// TIA Portal V17 export
// export: Created 2025-04-09T08:03:29.2675501Z, ExportSetting WithDefaults, DisplayName Totally Integrated Automation Portal, DisplayVersion V17 Update 8, DisplayName TIA Portal Openness, DisplayVersion V17 Update 8, DisplayName TIA Portal Version Control Interface, DisplayVersion V17, DisplayName SINAMICS Startdrive Advanced, DisplayVersion V17 SP2, DisplayName SINAMICS Startdrive G110M, G120, G120C, G120D, G120P, G115D, DisplayVersion V17 SP2, DisplayName SINAMICS Startdrive G130, G150, S120, S150, SINAMICS MV, S210, DisplayVersion V17 SP2, DisplayName STEP 7 Professional, DisplayVersion V17 Update 8, DisplayName SINUMERIK ONE STEP 7 Toolbox, DisplayVersion V17 Update 12, DisplayName SINUMERIK ONE PLC Basic Program Plus, DisplayVersion V17 Update 12, DisplayName SINUMERIK 840D sl STEP 7 Toolbox, DisplayVersion V17 Update 12, DisplayName STEP 7 Safety, DisplayVersion V17 Update 6, DisplayName WinCC Advanced, DisplayVersion V17 Update 8
FUNCTION "FC16012_METHOD_CALLS_U01_STA3_COAXIAL" : Void   // FC16012, LAD
{ S7_Optimized_Access := 'TRUE' }
VERSION : 0.1
// PC status values:
// 0-> Idle
// 1-> LaserCalibrating
// 2-> NozzleCalibrating
// 3-> JetCalibrating
// 4-> CladdingCalibrating
// 5-> NozzleAnalysis
// 6-> JetAnalysis
// 7-> CladdingAnalysis
// -1-> Error
// stored: AutoNumber false, IsIECCheckEnabled false, SetENOAutomatically false, UDAEnableTagReadback false
   VAR_TEMP
      AUX_WSTRING_PART_ID_STA3 : WString;
      AUX_WCHARS : Array[0..63] of WChar;
      index : Int;
      ALARM_AUX : Bool;
   END_VAR
   VAR CONSTANT
      VERSIONS_MAJOR : UInt;
      VERSIONS_MINOR : UInt;
      FC_NUMBER : DInt := 16012;
   END_VAR
   VAR_TEMP   // added for the SCL form of the ladder/FBD networks
      _w1 : Bool;
      _w2 : Bool;
   END_VAR
BEGIN

REGION Network 1 (SCL): TRANSFORM TO WCHARS
   FOR #index := 0 TO 63 DO
       #AUX_WCHARS[#index] := CHAR_TO_WCHAR("DB8000_PART_STATUS".UNIT_01.STATION_3.PART_A.PART_ID[#index]);
   END_FOR;
END_REGION

REGION Network 2: TRANSFORM TO WSTRING
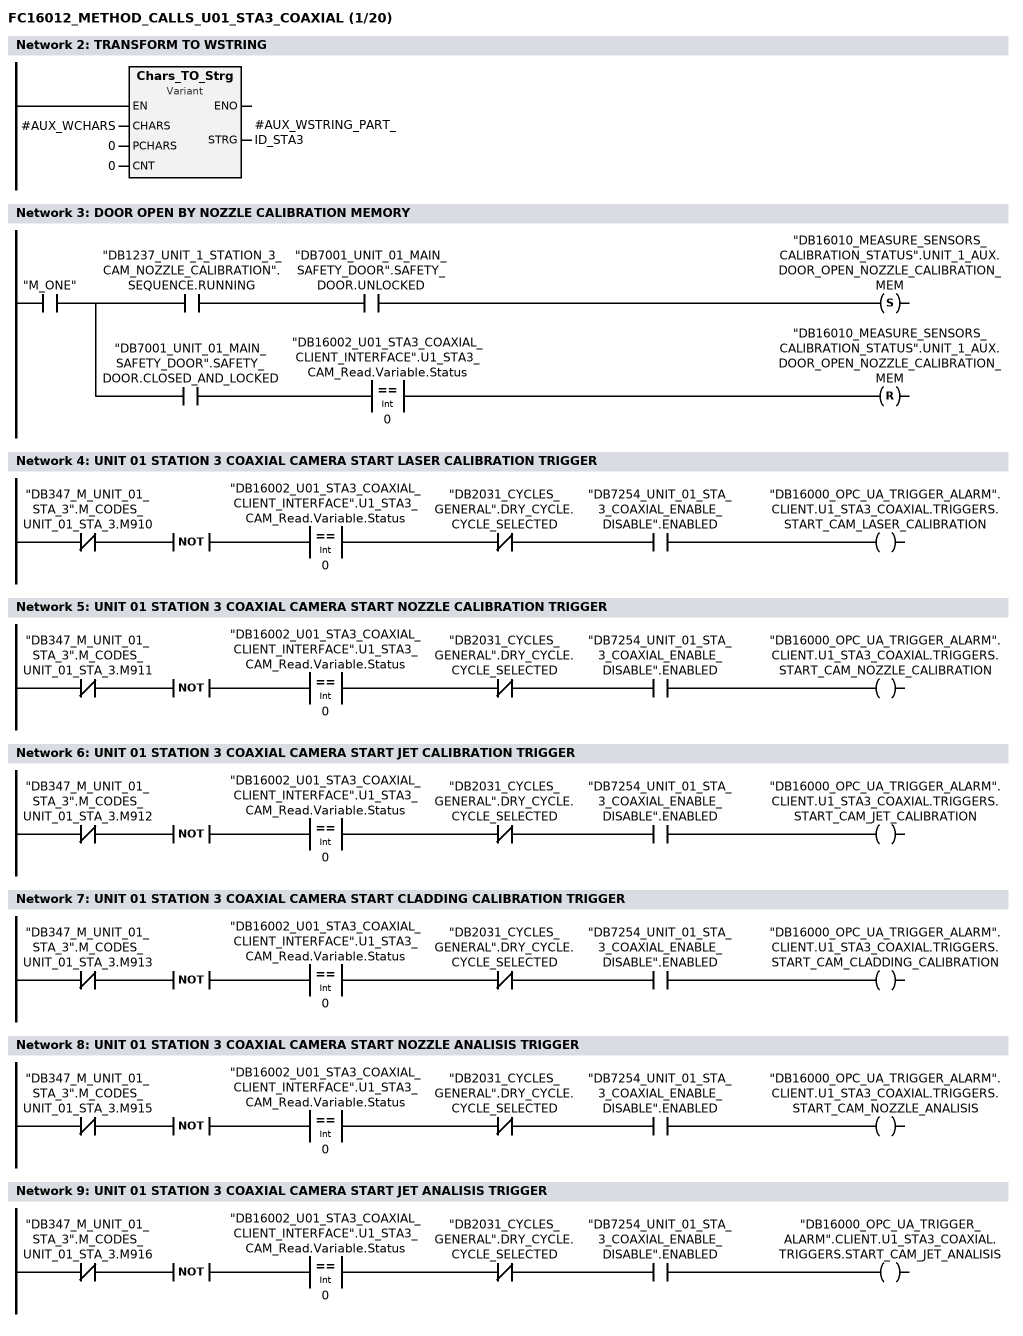
   RUNG wire#powerrail
      { S7_Templates := "[ptr_type := Variant, str_type := WString]" } Chars_TO_Strg(Chars := #AUX_WCHARS, pChars := 0, Cnt := 0, Strg => #AUX_WSTRING_PART_ID_STA3)
   END_RUNG
   // the same network as SCL:
   Chars_TO_Strg(Chars := #AUX_WCHARS, pChars := 0, Cnt := 0, Strg => #AUX_WSTRING_PART_ID_STA3);
END_REGION

REGION Network 3: DOOR OPEN BY NOZZLE CALIBRATION MEMORY
   RUNG wire#powerrail
      Contact( "M_ONE" )
      wire#w1
      Contact( "DB1237_UNIT_1_STATION_3_CAM_NOZZLE_CALIBRATION".SEQUENCE.RUNNING )
      Contact( "DB7001_UNIT_01_MAIN_SAFETY_DOOR".SAFETY_DOOR.UNLOCKED )
      S_Coil( "DB16010_MEASURE_SENSORS_CALIBRATION_STATUS".UNIT_1_AUX.DOOR_OPEN_NOZZLE_CALIBRATION_MEM )
   END_RUNG
   RUNG wire#w1
      Contact( "DB7001_UNIT_01_MAIN_SAFETY_DOOR".SAFETY_DOOR.CLOSED_AND_LOCKED )
      { S7_Templates := "SrcType := Int" } EQ_Contact(in1 := "DB16002_U01_STA3_COAXIAL_CLIENT_INTERFACE".U1_STA3_CAM_Read.Variable.Status, in2 := 0)
      R_Coil( "DB16010_MEASURE_SENSORS_CALIBRATION_STATUS".UNIT_1_AUX.DOOR_OPEN_NOZZLE_CALIBRATION_MEM )
   END_RUNG
   // the same network as SCL:
   IF "M_ONE" AND "DB1237_UNIT_1_STATION_3_CAM_NOZZLE_CALIBRATION".SEQUENCE.RUNNING AND "DB7001_UNIT_01_MAIN_SAFETY_DOOR".SAFETY_DOOR.UNLOCKED THEN
       "DB16010_MEASURE_SENSORS_CALIBRATION_STATUS".UNIT_1_AUX.DOOR_OPEN_NOZZLE_CALIBRATION_MEM := TRUE;
   END_IF;
   IF "M_ONE" AND "DB7001_UNIT_01_MAIN_SAFETY_DOOR".SAFETY_DOOR.CLOSED_AND_LOCKED AND ("DB16002_U01_STA3_COAXIAL_CLIENT_INTERFACE".U1_STA3_CAM_Read.Variable.Status = 0) THEN
       "DB16010_MEASURE_SENSORS_CALIBRATION_STATUS".UNIT_1_AUX.DOOR_OPEN_NOZZLE_CALIBRATION_MEM := FALSE;
   END_IF;
END_REGION

REGION Network 4: UNIT 01 STATION 3 COAXIAL CAMERA START LASER CALIBRATION TRIGGER
   RUNG wire#powerrail
      I_Contact( "DB347_M_UNIT_01_STA_3".M_CODES_UNIT_01_STA_3.M910 )
      Not()
      { S7_Templates := "SrcType := Int" } EQ_Contact(in1 := "DB16002_U01_STA3_COAXIAL_CLIENT_INTERFACE".U1_STA3_CAM_Read.Variable.Status, in2 := 0)
      I_Contact( "DB2031_CYCLES_GENERAL".DRY_CYCLE.CYCLE_SELECTED )
      Contact( "DB7254_UNIT_01_STA_3_COAXIAL_ENABLE_DISABLE".ENABLED )
      Coil( "DB16000_OPC_UA_TRIGGER_ALARM".CLIENT.U1_STA3_COAXIAL.TRIGGERS.START_CAM_LASER_CALIBRATION )
   END_RUNG
   // the same network as SCL:
   "DB16000_OPC_UA_TRIGGER_ALARM".CLIENT.U1_STA3_COAXIAL.TRIGGERS.START_CAM_LASER_CALIBRATION := NOT (NOT "DB347_M_UNIT_01_STA_3".M_CODES_UNIT_01_STA_3.M910) AND ("DB16002_U01_STA3_COAXIAL_CLIENT_INTERFACE".U1_STA3_CAM_Read.Variable.Status = 0) AND NOT "DB2031_CYCLES_GENERAL".DRY_CYCLE.CYCLE_SELECTED AND "DB7254_UNIT_01_STA_3_COAXIAL_ENABLE_DISABLE".ENABLED;
END_REGION

REGION Network 5: UNIT 01 STATION 3 COAXIAL CAMERA START NOZZLE CALIBRATION TRIGGER
   RUNG wire#powerrail
      I_Contact( "DB347_M_UNIT_01_STA_3".M_CODES_UNIT_01_STA_3.M911 )
      Not()
      { S7_Templates := "SrcType := Int" } EQ_Contact(in1 := "DB16002_U01_STA3_COAXIAL_CLIENT_INTERFACE".U1_STA3_CAM_Read.Variable.Status, in2 := 0)
      I_Contact( "DB2031_CYCLES_GENERAL".DRY_CYCLE.CYCLE_SELECTED )
      Contact( "DB7254_UNIT_01_STA_3_COAXIAL_ENABLE_DISABLE".ENABLED )
      Coil( "DB16000_OPC_UA_TRIGGER_ALARM".CLIENT.U1_STA3_COAXIAL.TRIGGERS.START_CAM_NOZZLE_CALIBRATION )
   END_RUNG
   // the same network as SCL:
   "DB16000_OPC_UA_TRIGGER_ALARM".CLIENT.U1_STA3_COAXIAL.TRIGGERS.START_CAM_NOZZLE_CALIBRATION := NOT (NOT "DB347_M_UNIT_01_STA_3".M_CODES_UNIT_01_STA_3.M911) AND ("DB16002_U01_STA3_COAXIAL_CLIENT_INTERFACE".U1_STA3_CAM_Read.Variable.Status = 0) AND NOT "DB2031_CYCLES_GENERAL".DRY_CYCLE.CYCLE_SELECTED AND "DB7254_UNIT_01_STA_3_COAXIAL_ENABLE_DISABLE".ENABLED;
END_REGION

REGION Network 6: UNIT 01 STATION 3 COAXIAL CAMERA START JET CALIBRATION TRIGGER
   RUNG wire#powerrail
      I_Contact( "DB347_M_UNIT_01_STA_3".M_CODES_UNIT_01_STA_3.M912 )
      Not()
      { S7_Templates := "SrcType := Int" } EQ_Contact(in1 := "DB16002_U01_STA3_COAXIAL_CLIENT_INTERFACE".U1_STA3_CAM_Read.Variable.Status, in2 := 0)
      I_Contact( "DB2031_CYCLES_GENERAL".DRY_CYCLE.CYCLE_SELECTED )
      Contact( "DB7254_UNIT_01_STA_3_COAXIAL_ENABLE_DISABLE".ENABLED )
      Coil( "DB16000_OPC_UA_TRIGGER_ALARM".CLIENT.U1_STA3_COAXIAL.TRIGGERS.START_CAM_JET_CALIBRATION )
   END_RUNG
   // the same network as SCL:
   "DB16000_OPC_UA_TRIGGER_ALARM".CLIENT.U1_STA3_COAXIAL.TRIGGERS.START_CAM_JET_CALIBRATION := NOT (NOT "DB347_M_UNIT_01_STA_3".M_CODES_UNIT_01_STA_3.M912) AND ("DB16002_U01_STA3_COAXIAL_CLIENT_INTERFACE".U1_STA3_CAM_Read.Variable.Status = 0) AND NOT "DB2031_CYCLES_GENERAL".DRY_CYCLE.CYCLE_SELECTED AND "DB7254_UNIT_01_STA_3_COAXIAL_ENABLE_DISABLE".ENABLED;
END_REGION

REGION Network 7: UNIT 01 STATION 3 COAXIAL CAMERA START CLADDING CALIBRATION TRIGGER
   RUNG wire#powerrail
      I_Contact( "DB347_M_UNIT_01_STA_3".M_CODES_UNIT_01_STA_3.M913 )
      Not()
      { S7_Templates := "SrcType := Int" } EQ_Contact(in1 := "DB16002_U01_STA3_COAXIAL_CLIENT_INTERFACE".U1_STA3_CAM_Read.Variable.Status, in2 := 0)
      I_Contact( "DB2031_CYCLES_GENERAL".DRY_CYCLE.CYCLE_SELECTED )
      Contact( "DB7254_UNIT_01_STA_3_COAXIAL_ENABLE_DISABLE".ENABLED )
      Coil( "DB16000_OPC_UA_TRIGGER_ALARM".CLIENT.U1_STA3_COAXIAL.TRIGGERS.START_CAM_CLADDING_CALIBRATION )
   END_RUNG
   // the same network as SCL:
   "DB16000_OPC_UA_TRIGGER_ALARM".CLIENT.U1_STA3_COAXIAL.TRIGGERS.START_CAM_CLADDING_CALIBRATION := NOT (NOT "DB347_M_UNIT_01_STA_3".M_CODES_UNIT_01_STA_3.M913) AND ("DB16002_U01_STA3_COAXIAL_CLIENT_INTERFACE".U1_STA3_CAM_Read.Variable.Status = 0) AND NOT "DB2031_CYCLES_GENERAL".DRY_CYCLE.CYCLE_SELECTED AND "DB7254_UNIT_01_STA_3_COAXIAL_ENABLE_DISABLE".ENABLED;
END_REGION

REGION Network 8: UNIT 01 STATION 3 COAXIAL CAMERA START NOZZLE ANALISIS TRIGGER
   RUNG wire#powerrail
      I_Contact( "DB347_M_UNIT_01_STA_3".M_CODES_UNIT_01_STA_3.M915 )
      Not()
      { S7_Templates := "SrcType := Int" } EQ_Contact(in1 := "DB16002_U01_STA3_COAXIAL_CLIENT_INTERFACE".U1_STA3_CAM_Read.Variable.Status, in2 := 0)
      I_Contact( "DB2031_CYCLES_GENERAL".DRY_CYCLE.CYCLE_SELECTED )
      Contact( "DB7254_UNIT_01_STA_3_COAXIAL_ENABLE_DISABLE".ENABLED )
      Coil( "DB16000_OPC_UA_TRIGGER_ALARM".CLIENT.U1_STA3_COAXIAL.TRIGGERS.START_CAM_NOZZLE_ANALISIS )
   END_RUNG
   // the same network as SCL:
   "DB16000_OPC_UA_TRIGGER_ALARM".CLIENT.U1_STA3_COAXIAL.TRIGGERS.START_CAM_NOZZLE_ANALISIS := NOT (NOT "DB347_M_UNIT_01_STA_3".M_CODES_UNIT_01_STA_3.M915) AND ("DB16002_U01_STA3_COAXIAL_CLIENT_INTERFACE".U1_STA3_CAM_Read.Variable.Status = 0) AND NOT "DB2031_CYCLES_GENERAL".DRY_CYCLE.CYCLE_SELECTED AND "DB7254_UNIT_01_STA_3_COAXIAL_ENABLE_DISABLE".ENABLED;
END_REGION

REGION Network 9: UNIT 01 STATION 3 COAXIAL CAMERA START JET ANALISIS TRIGGER
   RUNG wire#powerrail
      I_Contact( "DB347_M_UNIT_01_STA_3".M_CODES_UNIT_01_STA_3.M916 )
      Not()
      { S7_Templates := "SrcType := Int" } EQ_Contact(in1 := "DB16002_U01_STA3_COAXIAL_CLIENT_INTERFACE".U1_STA3_CAM_Read.Variable.Status, in2 := 0)
      I_Contact( "DB2031_CYCLES_GENERAL".DRY_CYCLE.CYCLE_SELECTED )
      Contact( "DB7254_UNIT_01_STA_3_COAXIAL_ENABLE_DISABLE".ENABLED )
      Coil( "DB16000_OPC_UA_TRIGGER_ALARM".CLIENT.U1_STA3_COAXIAL.TRIGGERS.START_CAM_JET_ANALISIS )
   END_RUNG
   // the same network as SCL:
   "DB16000_OPC_UA_TRIGGER_ALARM".CLIENT.U1_STA3_COAXIAL.TRIGGERS.START_CAM_JET_ANALISIS := NOT (NOT "DB347_M_UNIT_01_STA_3".M_CODES_UNIT_01_STA_3.M916) AND ("DB16002_U01_STA3_COAXIAL_CLIENT_INTERFACE".U1_STA3_CAM_Read.Variable.Status = 0) AND NOT "DB2031_CYCLES_GENERAL".DRY_CYCLE.CYCLE_SELECTED AND "DB7254_UNIT_01_STA_3_COAXIAL_ENABLE_DISABLE".ENABLED;
END_REGION

REGION Network 10: UNIT 01 STATION 3 COAXIAL CAMERA START CLADDING ANALISIS TRIGGER
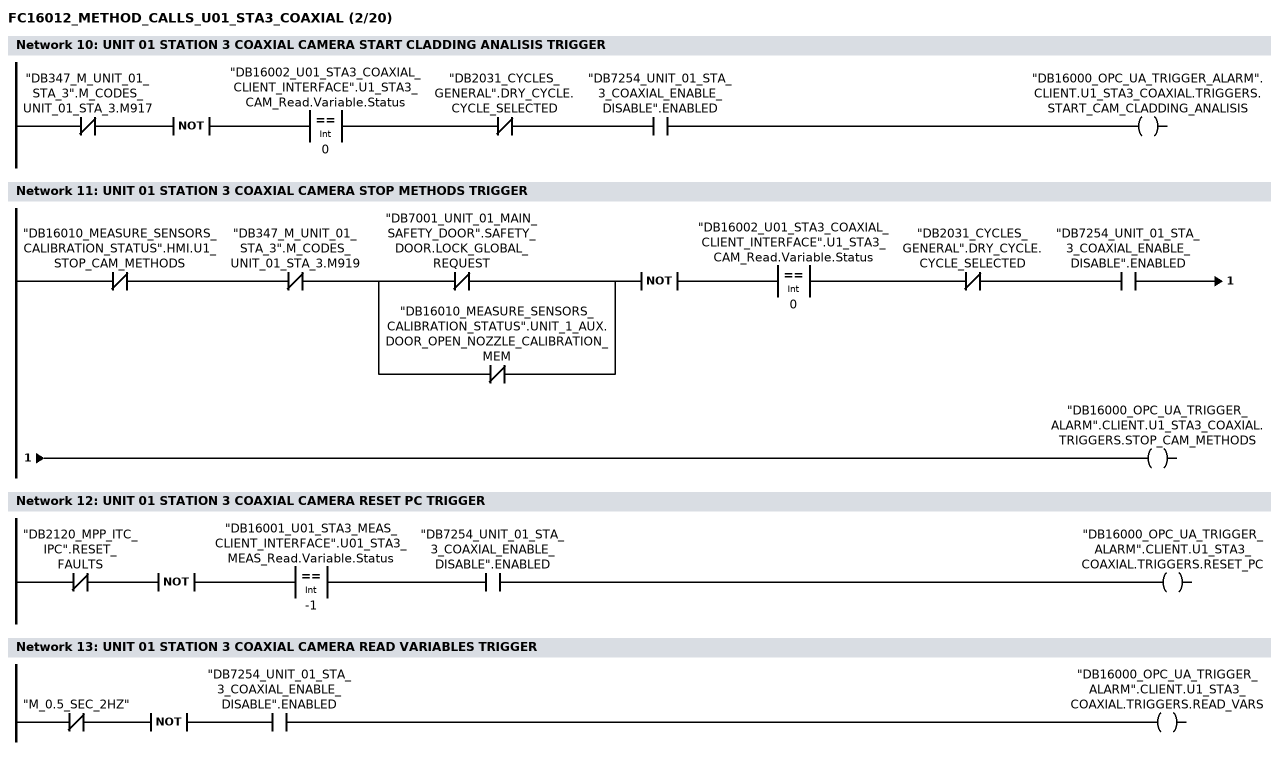
   RUNG wire#powerrail
      I_Contact( "DB347_M_UNIT_01_STA_3".M_CODES_UNIT_01_STA_3.M917 )
      Not()
      { S7_Templates := "SrcType := Int" } EQ_Contact(in1 := "DB16002_U01_STA3_COAXIAL_CLIENT_INTERFACE".U1_STA3_CAM_Read.Variable.Status, in2 := 0)
      I_Contact( "DB2031_CYCLES_GENERAL".DRY_CYCLE.CYCLE_SELECTED )
      Contact( "DB7254_UNIT_01_STA_3_COAXIAL_ENABLE_DISABLE".ENABLED )
      Coil( "DB16000_OPC_UA_TRIGGER_ALARM".CLIENT.U1_STA3_COAXIAL.TRIGGERS.START_CAM_CLADDING_ANALISIS )
   END_RUNG
   // the same network as SCL:
   "DB16000_OPC_UA_TRIGGER_ALARM".CLIENT.U1_STA3_COAXIAL.TRIGGERS.START_CAM_CLADDING_ANALISIS := NOT (NOT "DB347_M_UNIT_01_STA_3".M_CODES_UNIT_01_STA_3.M917) AND ("DB16002_U01_STA3_COAXIAL_CLIENT_INTERFACE".U1_STA3_CAM_Read.Variable.Status = 0) AND NOT "DB2031_CYCLES_GENERAL".DRY_CYCLE.CYCLE_SELECTED AND "DB7254_UNIT_01_STA_3_COAXIAL_ENABLE_DISABLE".ENABLED;
END_REGION

REGION Network 11: UNIT 01 STATION 3 COAXIAL CAMERA STOP METHODS TRIGGER
   RUNG wire#powerrail
      I_Contact( "DB16010_MEASURE_SENSORS_CALIBRATION_STATUS".HMI.U1_STOP_CAM_METHODS )
      I_Contact( "DB347_M_UNIT_01_STA_3".M_CODES_UNIT_01_STA_3.M919 )
      wire#w1
      I_Contact( "DB7001_UNIT_01_MAIN_SAFETY_DOOR".SAFETY_DOOR.LOCK_GLOBAL_REQUEST )
      wire#w2
      Not()
      { S7_Templates := "SrcType := Int" } EQ_Contact(in1 := "DB16002_U01_STA3_COAXIAL_CLIENT_INTERFACE".U1_STA3_CAM_Read.Variable.Status, in2 := 0)
      I_Contact( "DB2031_CYCLES_GENERAL".DRY_CYCLE.CYCLE_SELECTED )
      Contact( "DB7254_UNIT_01_STA_3_COAXIAL_ENABLE_DISABLE".ENABLED )
      Coil( "DB16000_OPC_UA_TRIGGER_ALARM".CLIENT.U1_STA3_COAXIAL.TRIGGERS.STOP_CAM_METHODS )
   END_RUNG
   RUNG wire#w1
      I_Contact( "DB16010_MEASURE_SENSORS_CALIBRATION_STATUS".UNIT_1_AUX.DOOR_OPEN_NOZZLE_CALIBRATION_MEM )
   END_RUNG wire#w2
   // the same network as SCL:
   "DB16000_OPC_UA_TRIGGER_ALARM".CLIENT.U1_STA3_COAXIAL.TRIGGERS.STOP_CAM_METHODS := NOT (NOT "DB16010_MEASURE_SENSORS_CALIBRATION_STATUS".HMI.U1_STOP_CAM_METHODS AND NOT "DB347_M_UNIT_01_STA_3".M_CODES_UNIT_01_STA_3.M919 AND (NOT "DB7001_UNIT_01_MAIN_SAFETY_DOOR".SAFETY_DOOR.LOCK_GLOBAL_REQUEST OR NOT "DB16010_MEASURE_SENSORS_CALIBRATION_STATUS".UNIT_1_AUX.DOOR_OPEN_NOZZLE_CALIBRATION_MEM)) AND ("DB16002_U01_STA3_COAXIAL_CLIENT_INTERFACE".U1_STA3_CAM_Read.Variable.Status = 0) AND NOT "DB2031_CYCLES_GENERAL".DRY_CYCLE.CYCLE_SELECTED AND "DB7254_UNIT_01_STA_3_COAXIAL_ENABLE_DISABLE".ENABLED;
END_REGION

REGION Network 12: UNIT 01 STATION 3 COAXIAL CAMERA RESET PC TRIGGER
   RUNG wire#powerrail
      I_Contact( "DB2120_MPP_ITC_IPC".RESET_FAULTS )
      Not()
      { S7_Templates := "SrcType := Int" } EQ_Contact(in1 := "DB16001_U01_STA3_MEAS_CLIENT_INTERFACE".U01_STA3_MEAS_Read.Variable.Status, in2 := -1)
      Contact( "DB7254_UNIT_01_STA_3_COAXIAL_ENABLE_DISABLE".ENABLED )
      Coil( "DB16000_OPC_UA_TRIGGER_ALARM".CLIENT.U1_STA3_COAXIAL.TRIGGERS.RESET_PC )
   END_RUNG
   // the same network as SCL:
   "DB16000_OPC_UA_TRIGGER_ALARM".CLIENT.U1_STA3_COAXIAL.TRIGGERS.RESET_PC := NOT (NOT "DB2120_MPP_ITC_IPC".RESET_FAULTS) AND ("DB16001_U01_STA3_MEAS_CLIENT_INTERFACE".U01_STA3_MEAS_Read.Variable.Status = (-1)) AND "DB7254_UNIT_01_STA_3_COAXIAL_ENABLE_DISABLE".ENABLED;
END_REGION

REGION Network 13: UNIT 01 STATION 3 COAXIAL CAMERA READ VARIABLES TRIGGER
   RUNG wire#powerrail
      I_Contact( "M_0.5_SEC_2HZ" )
      Not()
      Contact( "DB7254_UNIT_01_STA_3_COAXIAL_ENABLE_DISABLE".ENABLED )
      Coil( "DB16000_OPC_UA_TRIGGER_ALARM".CLIENT.U1_STA3_COAXIAL.TRIGGERS.READ_VARS )
   END_RUNG
   // the same network as SCL:
   "DB16000_OPC_UA_TRIGGER_ALARM".CLIENT.U1_STA3_COAXIAL.TRIGGERS.READ_VARS := NOT (NOT "M_0.5_SEC_2HZ") AND "DB7254_UNIT_01_STA_3_COAXIAL_ENABLE_DISABLE".ENABLED;
END_REGION

REGION Network 14: UNIT 01 STATION 3 COAXIAL CAMERA START LASER CALIBRATION TRIGGER CALL
   // CAMBIAR POR EL METODO CORRECTO
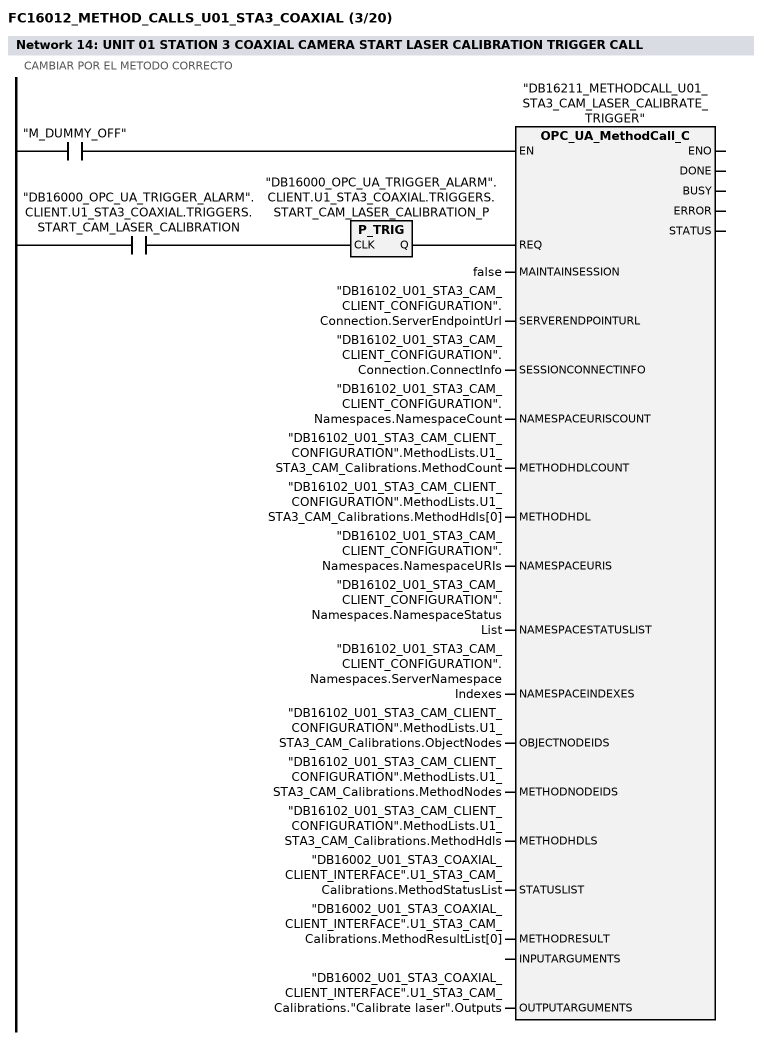
   RUNG wire#powerrail
      Contact( "M_DUMMY_OFF" )
      "DB16211_METHODCALL_U01_STA3_CAM_LASER_CALIBRATE_TRIGGER".OPC_UA_MethodCall_C(REQ := wire#w1, MaintainSession := false, ServerEndpointUrl := "DB16102_U01_STA3_CAM_CLIENT_CONFIGURATION".Connection.ServerEndpointUrl, SessionConnectInfo := "DB16102_U01_STA3_CAM_CLIENT_CONFIGURATION".Connection.ConnectInfo, NamespaceUrisCount := "DB16102_U01_STA3_CAM_CLIENT_CONFIGURATION".Namespaces.NamespaceCount, MethodHdlCount := "DB16102_U01_STA3_CAM_CLIENT_CONFIGURATION".MethodLists.U1_STA3_CAM_Calibrations.MethodCount, MethodHdl := "DB16102_U01_STA3_CAM_CLIENT_CONFIGURATION".MethodLists.U1_STA3_CAM_Calibrations.MethodHdls[0], NamespaceUris := "DB16102_U01_STA3_CAM_CLIENT_CONFIGURATION".Namespaces.NamespaceURIs, NamespaceStatusList := "DB16102_U01_STA3_CAM_CLIENT_CONFIGURATION".Namespaces.NamespaceStatusList, NamespaceIndexes := "DB16102_U01_STA3_CAM_CLIENT_CONFIGURATION".Namespaces.ServerNamespaceIndexes, ObjectNodeIDs := "DB16102_U01_STA3_CAM_CLIENT_CONFIGURATION".MethodLists.U1_STA3_CAM_Calibrations.ObjectNodes, MethodNodeIDs := "DB16102_U01_STA3_CAM_CLIENT_CONFIGURATION".MethodLists.U1_STA3_CAM_Calibrations.MethodNodes, MethodHdls := "DB16102_U01_STA3_CAM_CLIENT_CONFIGURATION".MethodLists.U1_STA3_CAM_Calibrations.MethodHdls, StatusList := "DB16002_U01_STA3_COAXIAL_CLIENT_INTERFACE".U1_STA3_CAM_Calibrations.MethodStatusList, MethodResult := "DB16002_U01_STA3_COAXIAL_CLIENT_INTERFACE".U1_STA3_CAM_Calibrations.MethodResultList[0], InputArguments :=, OutputArguments := "DB16002_U01_STA3_COAXIAL_CLIENT_INTERFACE".U1_STA3_CAM_Calibrations."Calibrate laser".Outputs, Done =>, Busy =>, Error =>, Status =>)
   END_RUNG
   RUNG wire#powerrail
      Contact( "DB16000_OPC_UA_TRIGGER_ALARM".CLIENT.U1_STA3_COAXIAL.TRIGGERS.START_CAM_LASER_CALIBRATION )
      P_Trig( "DB16000_OPC_UA_TRIGGER_ALARM".CLIENT.U1_STA3_COAXIAL.TRIGGERS.START_CAM_LASER_CALIBRATION_P )
   END_RUNG wire#w1
   // the same network as SCL:
   #_w1 := "DB16000_OPC_UA_TRIGGER_ALARM".CLIENT.U1_STA3_COAXIAL.TRIGGERS.START_CAM_LASER_CALIBRATION AND NOT "DB16000_OPC_UA_TRIGGER_ALARM".CLIENT.U1_STA3_COAXIAL.TRIGGERS.START_CAM_LASER_CALIBRATION_P;   // rising edge
   "DB16000_OPC_UA_TRIGGER_ALARM".CLIENT.U1_STA3_COAXIAL.TRIGGERS.START_CAM_LASER_CALIBRATION_P := "DB16000_OPC_UA_TRIGGER_ALARM".CLIENT.U1_STA3_COAXIAL.TRIGGERS.START_CAM_LASER_CALIBRATION;
   IF "M_DUMMY_OFF" THEN
       "DB16211_METHODCALL_U01_STA3_CAM_LASER_CALIBRATE_TRIGGER"(REQ := #_w1,   // OPC_UA_MethodCall_C
                               MaintainSession := false,
                               ServerEndpointUrl := "DB16102_U01_STA3_CAM_CLIENT_CONFIGURATION".Connection.ServerEndpointUrl,
                               SessionConnectInfo := "DB16102_U01_STA3_CAM_CLIENT_CONFIGURATION".Connection.ConnectInfo,
                               NamespaceUrisCount := "DB16102_U01_STA3_CAM_CLIENT_CONFIGURATION".Namespaces.NamespaceCount,
                               MethodHdlCount := "DB16102_U01_STA3_CAM_CLIENT_CONFIGURATION".MethodLists.U1_STA3_CAM_Calibrations.MethodCount,
                               MethodHdl := "DB16102_U01_STA3_CAM_CLIENT_CONFIGURATION".MethodLists.U1_STA3_CAM_Calibrations.MethodHdls[0],
                               NamespaceUris := "DB16102_U01_STA3_CAM_CLIENT_CONFIGURATION".Namespaces.NamespaceURIs,
                               NamespaceStatusList := "DB16102_U01_STA3_CAM_CLIENT_CONFIGURATION".Namespaces.NamespaceStatusList,
                               NamespaceIndexes := "DB16102_U01_STA3_CAM_CLIENT_CONFIGURATION".Namespaces.ServerNamespaceIndexes,
                               ObjectNodeIDs := "DB16102_U01_STA3_CAM_CLIENT_CONFIGURATION".MethodLists.U1_STA3_CAM_Calibrations.ObjectNodes,
                               MethodNodeIDs := "DB16102_U01_STA3_CAM_CLIENT_CONFIGURATION".MethodLists.U1_STA3_CAM_Calibrations.MethodNodes,
                               MethodHdls := "DB16102_U01_STA3_CAM_CLIENT_CONFIGURATION".MethodLists.U1_STA3_CAM_Calibrations.MethodHdls,
                               StatusList := "DB16002_U01_STA3_COAXIAL_CLIENT_INTERFACE".U1_STA3_CAM_Calibrations.MethodStatusList,
                               MethodResult := "DB16002_U01_STA3_COAXIAL_CLIENT_INTERFACE".U1_STA3_CAM_Calibrations.MethodResultList[0],
                               OutputArguments := "DB16002_U01_STA3_COAXIAL_CLIENT_INTERFACE".U1_STA3_CAM_Calibrations."Calibrate laser".Outputs);
   END_IF;
END_REGION

REGION Network 15: UNIT 01 STATION 3 COAXIAL CAMERA START NOZZLE CALIBRATION TRIGGER CALL
   // CAMBIAR POR EL METODO CORRECTO
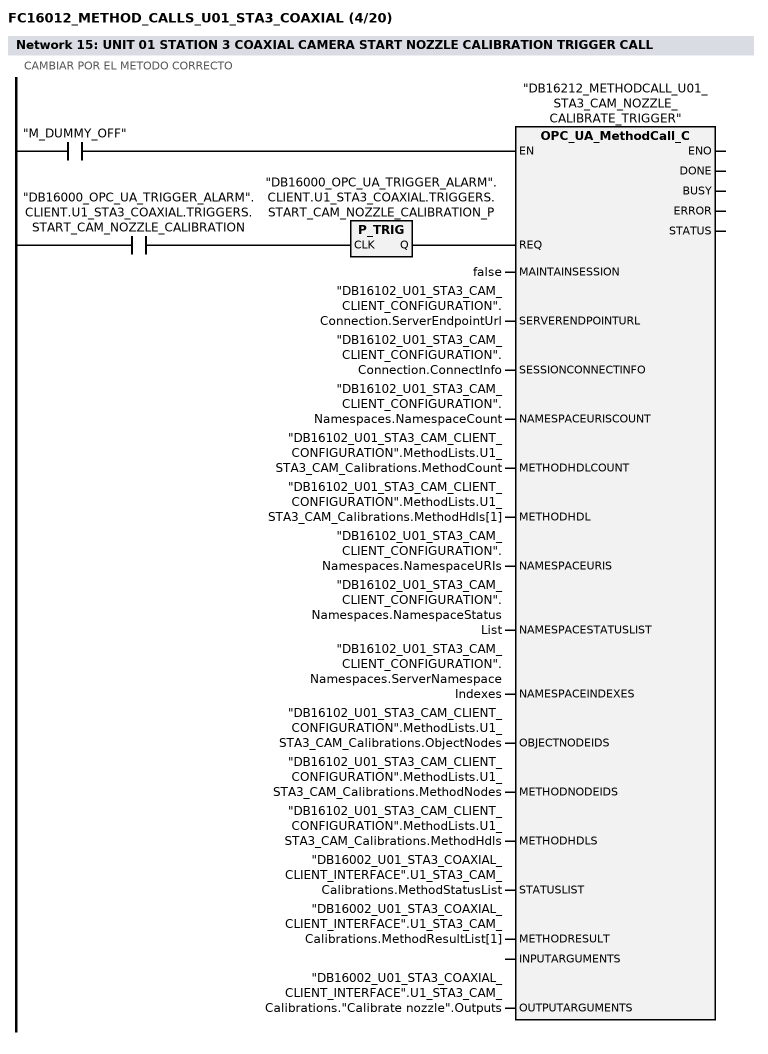
   RUNG wire#powerrail
      Contact( "M_DUMMY_OFF" )
      "DB16212_METHODCALL_U01_STA3_CAM_NOZZLE_CALIBRATE_TRIGGER".OPC_UA_MethodCall_C(REQ := wire#w1, MaintainSession := false, ServerEndpointUrl := "DB16102_U01_STA3_CAM_CLIENT_CONFIGURATION".Connection.ServerEndpointUrl, SessionConnectInfo := "DB16102_U01_STA3_CAM_CLIENT_CONFIGURATION".Connection.ConnectInfo, NamespaceUrisCount := "DB16102_U01_STA3_CAM_CLIENT_CONFIGURATION".Namespaces.NamespaceCount, MethodHdlCount := "DB16102_U01_STA3_CAM_CLIENT_CONFIGURATION".MethodLists.U1_STA3_CAM_Calibrations.MethodCount, MethodHdl := "DB16102_U01_STA3_CAM_CLIENT_CONFIGURATION".MethodLists.U1_STA3_CAM_Calibrations.MethodHdls[1], NamespaceUris := "DB16102_U01_STA3_CAM_CLIENT_CONFIGURATION".Namespaces.NamespaceURIs, NamespaceStatusList := "DB16102_U01_STA3_CAM_CLIENT_CONFIGURATION".Namespaces.NamespaceStatusList, NamespaceIndexes := "DB16102_U01_STA3_CAM_CLIENT_CONFIGURATION".Namespaces.ServerNamespaceIndexes, ObjectNodeIDs := "DB16102_U01_STA3_CAM_CLIENT_CONFIGURATION".MethodLists.U1_STA3_CAM_Calibrations.ObjectNodes, MethodNodeIDs := "DB16102_U01_STA3_CAM_CLIENT_CONFIGURATION".MethodLists.U1_STA3_CAM_Calibrations.MethodNodes, MethodHdls := "DB16102_U01_STA3_CAM_CLIENT_CONFIGURATION".MethodLists.U1_STA3_CAM_Calibrations.MethodHdls, StatusList := "DB16002_U01_STA3_COAXIAL_CLIENT_INTERFACE".U1_STA3_CAM_Calibrations.MethodStatusList, MethodResult := "DB16002_U01_STA3_COAXIAL_CLIENT_INTERFACE".U1_STA3_CAM_Calibrations.MethodResultList[1], InputArguments :=, OutputArguments := "DB16002_U01_STA3_COAXIAL_CLIENT_INTERFACE".U1_STA3_CAM_Calibrations."Calibrate nozzle".Outputs, Done =>, Busy =>, Error =>, Status =>)
   END_RUNG
   RUNG wire#powerrail
      Contact( "DB16000_OPC_UA_TRIGGER_ALARM".CLIENT.U1_STA3_COAXIAL.TRIGGERS.START_CAM_NOZZLE_CALIBRATION )
      P_Trig( "DB16000_OPC_UA_TRIGGER_ALARM".CLIENT.U1_STA3_COAXIAL.TRIGGERS.START_CAM_NOZZLE_CALIBRATION_P )
   END_RUNG wire#w1
   // the same network as SCL:
   #_w1 := "DB16000_OPC_UA_TRIGGER_ALARM".CLIENT.U1_STA3_COAXIAL.TRIGGERS.START_CAM_NOZZLE_CALIBRATION AND NOT "DB16000_OPC_UA_TRIGGER_ALARM".CLIENT.U1_STA3_COAXIAL.TRIGGERS.START_CAM_NOZZLE_CALIBRATION_P;   // rising edge
   "DB16000_OPC_UA_TRIGGER_ALARM".CLIENT.U1_STA3_COAXIAL.TRIGGERS.START_CAM_NOZZLE_CALIBRATION_P := "DB16000_OPC_UA_TRIGGER_ALARM".CLIENT.U1_STA3_COAXIAL.TRIGGERS.START_CAM_NOZZLE_CALIBRATION;
   IF "M_DUMMY_OFF" THEN
       "DB16212_METHODCALL_U01_STA3_CAM_NOZZLE_CALIBRATE_TRIGGER"(REQ := #_w1,   // OPC_UA_MethodCall_C
                               MaintainSession := false,
                               ServerEndpointUrl := "DB16102_U01_STA3_CAM_CLIENT_CONFIGURATION".Connection.ServerEndpointUrl,
                               SessionConnectInfo := "DB16102_U01_STA3_CAM_CLIENT_CONFIGURATION".Connection.ConnectInfo,
                               NamespaceUrisCount := "DB16102_U01_STA3_CAM_CLIENT_CONFIGURATION".Namespaces.NamespaceCount,
                               MethodHdlCount := "DB16102_U01_STA3_CAM_CLIENT_CONFIGURATION".MethodLists.U1_STA3_CAM_Calibrations.MethodCount,
                               MethodHdl := "DB16102_U01_STA3_CAM_CLIENT_CONFIGURATION".MethodLists.U1_STA3_CAM_Calibrations.MethodHdls[1],
                               NamespaceUris := "DB16102_U01_STA3_CAM_CLIENT_CONFIGURATION".Namespaces.NamespaceURIs,
                               NamespaceStatusList := "DB16102_U01_STA3_CAM_CLIENT_CONFIGURATION".Namespaces.NamespaceStatusList,
                               NamespaceIndexes := "DB16102_U01_STA3_CAM_CLIENT_CONFIGURATION".Namespaces.ServerNamespaceIndexes,
                               ObjectNodeIDs := "DB16102_U01_STA3_CAM_CLIENT_CONFIGURATION".MethodLists.U1_STA3_CAM_Calibrations.ObjectNodes,
                               MethodNodeIDs := "DB16102_U01_STA3_CAM_CLIENT_CONFIGURATION".MethodLists.U1_STA3_CAM_Calibrations.MethodNodes,
                               MethodHdls := "DB16102_U01_STA3_CAM_CLIENT_CONFIGURATION".MethodLists.U1_STA3_CAM_Calibrations.MethodHdls,
                               StatusList := "DB16002_U01_STA3_COAXIAL_CLIENT_INTERFACE".U1_STA3_CAM_Calibrations.MethodStatusList,
                               MethodResult := "DB16002_U01_STA3_COAXIAL_CLIENT_INTERFACE".U1_STA3_CAM_Calibrations.MethodResultList[1],
                               OutputArguments := "DB16002_U01_STA3_COAXIAL_CLIENT_INTERFACE".U1_STA3_CAM_Calibrations."Calibrate nozzle".Outputs);
   END_IF;
END_REGION

REGION Network 16: UNIT 01 STATION 3 COAXIAL CAMERA START JET CALIBRATION TRIGGER CALL
   // CAMBIAR POR EL METODO CORRECTO
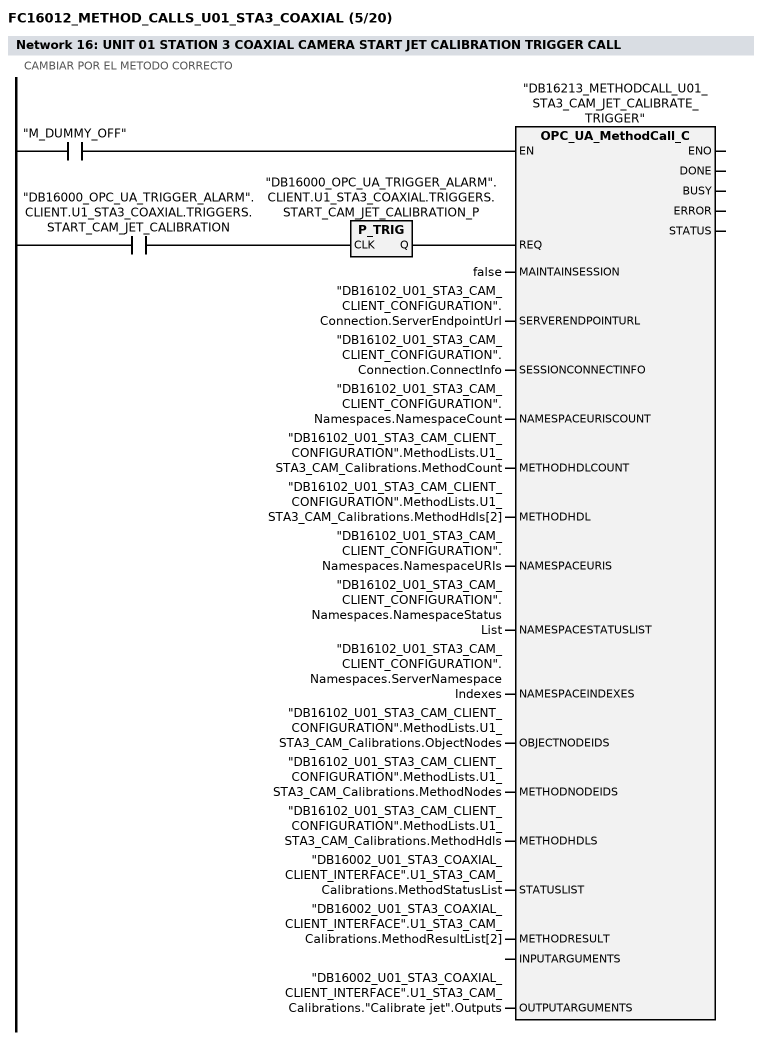
   RUNG wire#powerrail
      Contact( "M_DUMMY_OFF" )
      "DB16213_METHODCALL_U01_STA3_CAM_JET_CALIBRATE_TRIGGER".OPC_UA_MethodCall_C(REQ := wire#w1, MaintainSession := false, ServerEndpointUrl := "DB16102_U01_STA3_CAM_CLIENT_CONFIGURATION".Connection.ServerEndpointUrl, SessionConnectInfo := "DB16102_U01_STA3_CAM_CLIENT_CONFIGURATION".Connection.ConnectInfo, NamespaceUrisCount := "DB16102_U01_STA3_CAM_CLIENT_CONFIGURATION".Namespaces.NamespaceCount, MethodHdlCount := "DB16102_U01_STA3_CAM_CLIENT_CONFIGURATION".MethodLists.U1_STA3_CAM_Calibrations.MethodCount, MethodHdl := "DB16102_U01_STA3_CAM_CLIENT_CONFIGURATION".MethodLists.U1_STA3_CAM_Calibrations.MethodHdls[2], NamespaceUris := "DB16102_U01_STA3_CAM_CLIENT_CONFIGURATION".Namespaces.NamespaceURIs, NamespaceStatusList := "DB16102_U01_STA3_CAM_CLIENT_CONFIGURATION".Namespaces.NamespaceStatusList, NamespaceIndexes := "DB16102_U01_STA3_CAM_CLIENT_CONFIGURATION".Namespaces.ServerNamespaceIndexes, ObjectNodeIDs := "DB16102_U01_STA3_CAM_CLIENT_CONFIGURATION".MethodLists.U1_STA3_CAM_Calibrations.ObjectNodes, MethodNodeIDs := "DB16102_U01_STA3_CAM_CLIENT_CONFIGURATION".MethodLists.U1_STA3_CAM_Calibrations.MethodNodes, MethodHdls := "DB16102_U01_STA3_CAM_CLIENT_CONFIGURATION".MethodLists.U1_STA3_CAM_Calibrations.MethodHdls, StatusList := "DB16002_U01_STA3_COAXIAL_CLIENT_INTERFACE".U1_STA3_CAM_Calibrations.MethodStatusList, MethodResult := "DB16002_U01_STA3_COAXIAL_CLIENT_INTERFACE".U1_STA3_CAM_Calibrations.MethodResultList[2], InputArguments :=, OutputArguments := "DB16002_U01_STA3_COAXIAL_CLIENT_INTERFACE".U1_STA3_CAM_Calibrations."Calibrate jet".Outputs, Done =>, Busy =>, Error =>, Status =>)
   END_RUNG
   RUNG wire#powerrail
      Contact( "DB16000_OPC_UA_TRIGGER_ALARM".CLIENT.U1_STA3_COAXIAL.TRIGGERS.START_CAM_JET_CALIBRATION )
      P_Trig( "DB16000_OPC_UA_TRIGGER_ALARM".CLIENT.U1_STA3_COAXIAL.TRIGGERS.START_CAM_JET_CALIBRATION_P )
   END_RUNG wire#w1
   // the same network as SCL:
   #_w1 := "DB16000_OPC_UA_TRIGGER_ALARM".CLIENT.U1_STA3_COAXIAL.TRIGGERS.START_CAM_JET_CALIBRATION AND NOT "DB16000_OPC_UA_TRIGGER_ALARM".CLIENT.U1_STA3_COAXIAL.TRIGGERS.START_CAM_JET_CALIBRATION_P;   // rising edge
   "DB16000_OPC_UA_TRIGGER_ALARM".CLIENT.U1_STA3_COAXIAL.TRIGGERS.START_CAM_JET_CALIBRATION_P := "DB16000_OPC_UA_TRIGGER_ALARM".CLIENT.U1_STA3_COAXIAL.TRIGGERS.START_CAM_JET_CALIBRATION;
   IF "M_DUMMY_OFF" THEN
       "DB16213_METHODCALL_U01_STA3_CAM_JET_CALIBRATE_TRIGGER"(REQ := #_w1,   // OPC_UA_MethodCall_C
                               MaintainSession := false,
                               ServerEndpointUrl := "DB16102_U01_STA3_CAM_CLIENT_CONFIGURATION".Connection.ServerEndpointUrl,
                               SessionConnectInfo := "DB16102_U01_STA3_CAM_CLIENT_CONFIGURATION".Connection.ConnectInfo,
                               NamespaceUrisCount := "DB16102_U01_STA3_CAM_CLIENT_CONFIGURATION".Namespaces.NamespaceCount,
                               MethodHdlCount := "DB16102_U01_STA3_CAM_CLIENT_CONFIGURATION".MethodLists.U1_STA3_CAM_Calibrations.MethodCount,
                               MethodHdl := "DB16102_U01_STA3_CAM_CLIENT_CONFIGURATION".MethodLists.U1_STA3_CAM_Calibrations.MethodHdls[2],
                               NamespaceUris := "DB16102_U01_STA3_CAM_CLIENT_CONFIGURATION".Namespaces.NamespaceURIs,
                               NamespaceStatusList := "DB16102_U01_STA3_CAM_CLIENT_CONFIGURATION".Namespaces.NamespaceStatusList,
                               NamespaceIndexes := "DB16102_U01_STA3_CAM_CLIENT_CONFIGURATION".Namespaces.ServerNamespaceIndexes,
                               ObjectNodeIDs := "DB16102_U01_STA3_CAM_CLIENT_CONFIGURATION".MethodLists.U1_STA3_CAM_Calibrations.ObjectNodes,
                               MethodNodeIDs := "DB16102_U01_STA3_CAM_CLIENT_CONFIGURATION".MethodLists.U1_STA3_CAM_Calibrations.MethodNodes,
                               MethodHdls := "DB16102_U01_STA3_CAM_CLIENT_CONFIGURATION".MethodLists.U1_STA3_CAM_Calibrations.MethodHdls,
                               StatusList := "DB16002_U01_STA3_COAXIAL_CLIENT_INTERFACE".U1_STA3_CAM_Calibrations.MethodStatusList,
                               MethodResult := "DB16002_U01_STA3_COAXIAL_CLIENT_INTERFACE".U1_STA3_CAM_Calibrations.MethodResultList[2],
                               OutputArguments := "DB16002_U01_STA3_COAXIAL_CLIENT_INTERFACE".U1_STA3_CAM_Calibrations."Calibrate jet".Outputs);
   END_IF;
END_REGION

REGION Network 17: UNIT 01 STATION 3 COAXIAL CAMERA START CLADDING CALIBRATION TRIGGER CALL
   // CAMBIAR POR EL METODO CORRECTO
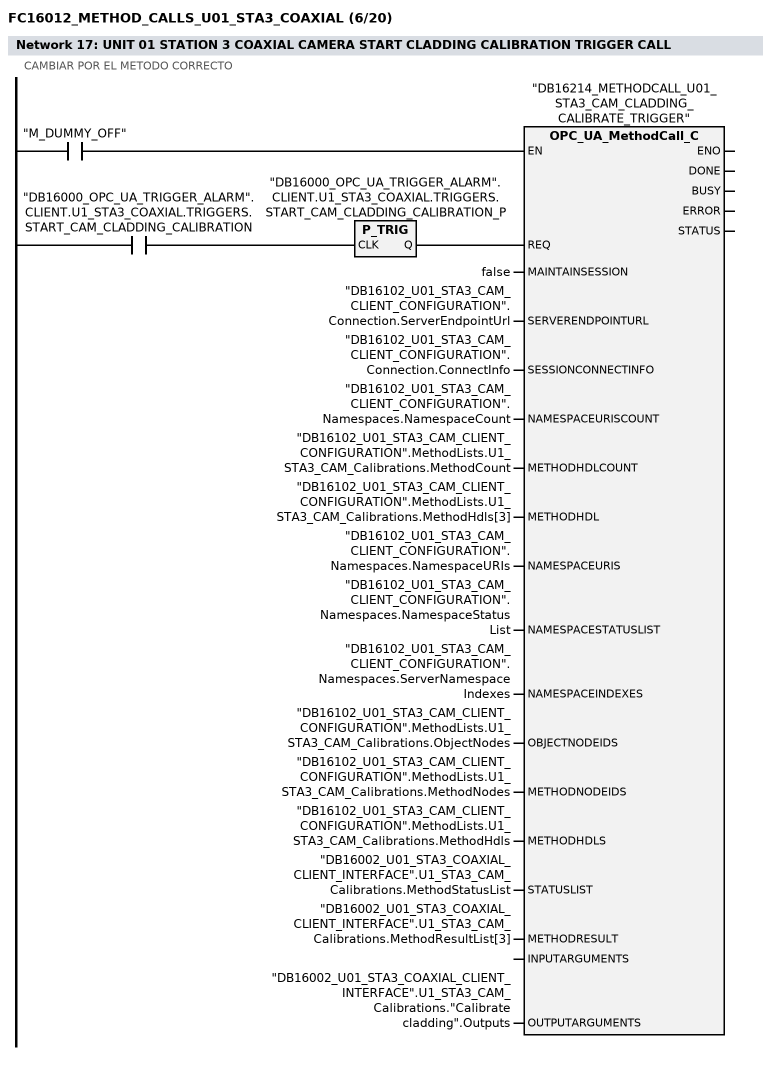
   RUNG wire#powerrail
      Contact( "M_DUMMY_OFF" )
      "DB16214_METHODCALL_U01_STA3_CAM_CLADDING_CALIBRATE_TRIGGER".OPC_UA_MethodCall_C(REQ := wire#w1, MaintainSession := false, ServerEndpointUrl := "DB16102_U01_STA3_CAM_CLIENT_CONFIGURATION".Connection.ServerEndpointUrl, SessionConnectInfo := "DB16102_U01_STA3_CAM_CLIENT_CONFIGURATION".Connection.ConnectInfo, NamespaceUrisCount := "DB16102_U01_STA3_CAM_CLIENT_CONFIGURATION".Namespaces.NamespaceCount, MethodHdlCount := "DB16102_U01_STA3_CAM_CLIENT_CONFIGURATION".MethodLists.U1_STA3_CAM_Calibrations.MethodCount, MethodHdl := "DB16102_U01_STA3_CAM_CLIENT_CONFIGURATION".MethodLists.U1_STA3_CAM_Calibrations.MethodHdls[3], NamespaceUris := "DB16102_U01_STA3_CAM_CLIENT_CONFIGURATION".Namespaces.NamespaceURIs, NamespaceStatusList := "DB16102_U01_STA3_CAM_CLIENT_CONFIGURATION".Namespaces.NamespaceStatusList, NamespaceIndexes := "DB16102_U01_STA3_CAM_CLIENT_CONFIGURATION".Namespaces.ServerNamespaceIndexes, ObjectNodeIDs := "DB16102_U01_STA3_CAM_CLIENT_CONFIGURATION".MethodLists.U1_STA3_CAM_Calibrations.ObjectNodes, MethodNodeIDs := "DB16102_U01_STA3_CAM_CLIENT_CONFIGURATION".MethodLists.U1_STA3_CAM_Calibrations.MethodNodes, MethodHdls := "DB16102_U01_STA3_CAM_CLIENT_CONFIGURATION".MethodLists.U1_STA3_CAM_Calibrations.MethodHdls, StatusList := "DB16002_U01_STA3_COAXIAL_CLIENT_INTERFACE".U1_STA3_CAM_Calibrations.MethodStatusList, MethodResult := "DB16002_U01_STA3_COAXIAL_CLIENT_INTERFACE".U1_STA3_CAM_Calibrations.MethodResultList[3], InputArguments :=, OutputArguments := "DB16002_U01_STA3_COAXIAL_CLIENT_INTERFACE".U1_STA3_CAM_Calibrations."Calibrate cladding".Outputs, Done =>, Busy =>, Error =>, Status =>)
   END_RUNG
   RUNG wire#powerrail
      Contact( "DB16000_OPC_UA_TRIGGER_ALARM".CLIENT.U1_STA3_COAXIAL.TRIGGERS.START_CAM_CLADDING_CALIBRATION )
      P_Trig( "DB16000_OPC_UA_TRIGGER_ALARM".CLIENT.U1_STA3_COAXIAL.TRIGGERS.START_CAM_CLADDING_CALIBRATION_P )
   END_RUNG wire#w1
   // the same network as SCL:
   #_w1 := "DB16000_OPC_UA_TRIGGER_ALARM".CLIENT.U1_STA3_COAXIAL.TRIGGERS.START_CAM_CLADDING_CALIBRATION AND NOT "DB16000_OPC_UA_TRIGGER_ALARM".CLIENT.U1_STA3_COAXIAL.TRIGGERS.START_CAM_CLADDING_CALIBRATION_P;   // rising edge
   "DB16000_OPC_UA_TRIGGER_ALARM".CLIENT.U1_STA3_COAXIAL.TRIGGERS.START_CAM_CLADDING_CALIBRATION_P := "DB16000_OPC_UA_TRIGGER_ALARM".CLIENT.U1_STA3_COAXIAL.TRIGGERS.START_CAM_CLADDING_CALIBRATION;
   IF "M_DUMMY_OFF" THEN
       "DB16214_METHODCALL_U01_STA3_CAM_CLADDING_CALIBRATE_TRIGGER"(REQ := #_w1,   // OPC_UA_MethodCall_C
                               MaintainSession := false,
                               ServerEndpointUrl := "DB16102_U01_STA3_CAM_CLIENT_CONFIGURATION".Connection.ServerEndpointUrl,
                               SessionConnectInfo := "DB16102_U01_STA3_CAM_CLIENT_CONFIGURATION".Connection.ConnectInfo,
                               NamespaceUrisCount := "DB16102_U01_STA3_CAM_CLIENT_CONFIGURATION".Namespaces.NamespaceCount,
                               MethodHdlCount := "DB16102_U01_STA3_CAM_CLIENT_CONFIGURATION".MethodLists.U1_STA3_CAM_Calibrations.MethodCount,
                               MethodHdl := "DB16102_U01_STA3_CAM_CLIENT_CONFIGURATION".MethodLists.U1_STA3_CAM_Calibrations.MethodHdls[3],
                               NamespaceUris := "DB16102_U01_STA3_CAM_CLIENT_CONFIGURATION".Namespaces.NamespaceURIs,
                               NamespaceStatusList := "DB16102_U01_STA3_CAM_CLIENT_CONFIGURATION".Namespaces.NamespaceStatusList,
                               NamespaceIndexes := "DB16102_U01_STA3_CAM_CLIENT_CONFIGURATION".Namespaces.ServerNamespaceIndexes,
                               ObjectNodeIDs := "DB16102_U01_STA3_CAM_CLIENT_CONFIGURATION".MethodLists.U1_STA3_CAM_Calibrations.ObjectNodes,
                               MethodNodeIDs := "DB16102_U01_STA3_CAM_CLIENT_CONFIGURATION".MethodLists.U1_STA3_CAM_Calibrations.MethodNodes,
                               MethodHdls := "DB16102_U01_STA3_CAM_CLIENT_CONFIGURATION".MethodLists.U1_STA3_CAM_Calibrations.MethodHdls,
                               StatusList := "DB16002_U01_STA3_COAXIAL_CLIENT_INTERFACE".U1_STA3_CAM_Calibrations.MethodStatusList,
                               MethodResult := "DB16002_U01_STA3_COAXIAL_CLIENT_INTERFACE".U1_STA3_CAM_Calibrations.MethodResultList[3],
                               OutputArguments := "DB16002_U01_STA3_COAXIAL_CLIENT_INTERFACE".U1_STA3_CAM_Calibrations."Calibrate cladding".Outputs);
   END_IF;
END_REGION

REGION Network 18: UNIT 01 STATION 3 COAXIAL CAMERA START NOZZLE ANALISIS TRIGGER CALL
   // CAMBIAR POR EL METODO CORRECTO
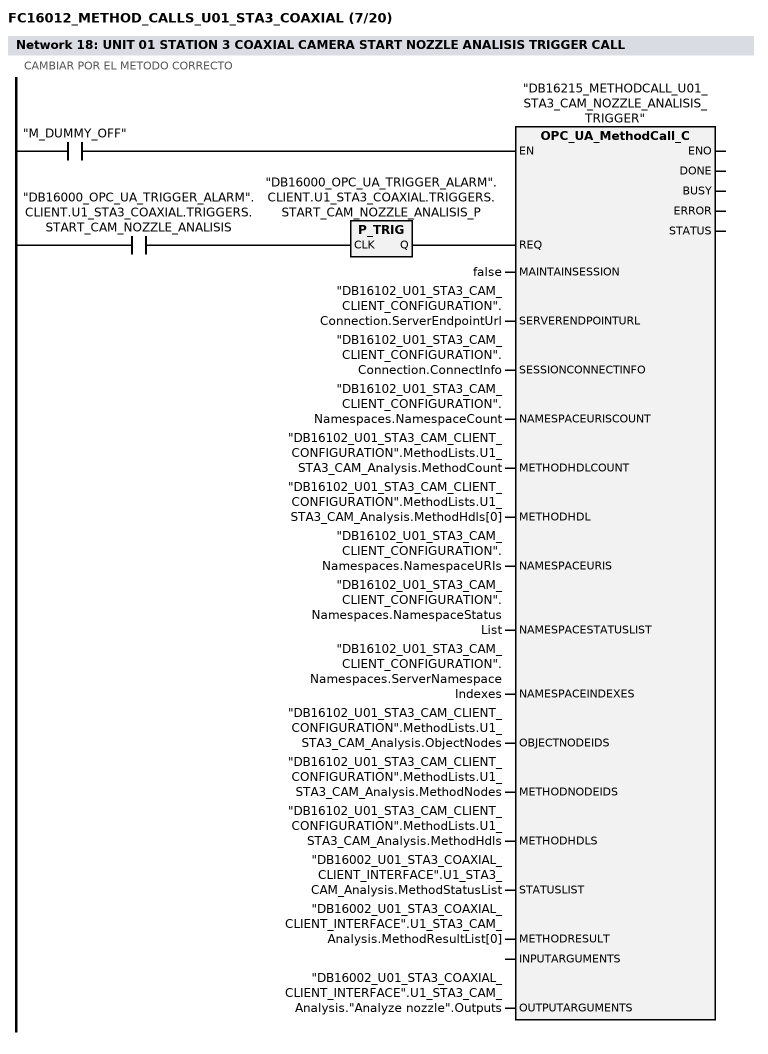
   RUNG wire#powerrail
      Contact( "M_DUMMY_OFF" )
      "DB16215_METHODCALL_U01_STA3_CAM_NOZZLE_ANALISIS_TRIGGER".OPC_UA_MethodCall_C(REQ := wire#w1, MaintainSession := false, ServerEndpointUrl := "DB16102_U01_STA3_CAM_CLIENT_CONFIGURATION".Connection.ServerEndpointUrl, SessionConnectInfo := "DB16102_U01_STA3_CAM_CLIENT_CONFIGURATION".Connection.ConnectInfo, NamespaceUrisCount := "DB16102_U01_STA3_CAM_CLIENT_CONFIGURATION".Namespaces.NamespaceCount, MethodHdlCount := "DB16102_U01_STA3_CAM_CLIENT_CONFIGURATION".MethodLists.U1_STA3_CAM_Analysis.MethodCount, MethodHdl := "DB16102_U01_STA3_CAM_CLIENT_CONFIGURATION".MethodLists.U1_STA3_CAM_Analysis.MethodHdls[0], NamespaceUris := "DB16102_U01_STA3_CAM_CLIENT_CONFIGURATION".Namespaces.NamespaceURIs, NamespaceStatusList := "DB16102_U01_STA3_CAM_CLIENT_CONFIGURATION".Namespaces.NamespaceStatusList, NamespaceIndexes := "DB16102_U01_STA3_CAM_CLIENT_CONFIGURATION".Namespaces.ServerNamespaceIndexes, ObjectNodeIDs := "DB16102_U01_STA3_CAM_CLIENT_CONFIGURATION".MethodLists.U1_STA3_CAM_Analysis.ObjectNodes, MethodNodeIDs := "DB16102_U01_STA3_CAM_CLIENT_CONFIGURATION".MethodLists.U1_STA3_CAM_Analysis.MethodNodes, MethodHdls := "DB16102_U01_STA3_CAM_CLIENT_CONFIGURATION".MethodLists.U1_STA3_CAM_Analysis.MethodHdls, StatusList := "DB16002_U01_STA3_COAXIAL_CLIENT_INTERFACE".U1_STA3_CAM_Analysis.MethodStatusList, MethodResult := "DB16002_U01_STA3_COAXIAL_CLIENT_INTERFACE".U1_STA3_CAM_Analysis.MethodResultList[0], InputArguments :=, OutputArguments := "DB16002_U01_STA3_COAXIAL_CLIENT_INTERFACE".U1_STA3_CAM_Analysis."Analyze nozzle".Outputs, Done =>, Busy =>, Error =>, Status =>)
   END_RUNG
   RUNG wire#powerrail
      Contact( "DB16000_OPC_UA_TRIGGER_ALARM".CLIENT.U1_STA3_COAXIAL.TRIGGERS.START_CAM_NOZZLE_ANALISIS )
      P_Trig( "DB16000_OPC_UA_TRIGGER_ALARM".CLIENT.U1_STA3_COAXIAL.TRIGGERS.START_CAM_NOZZLE_ANALISIS_P )
   END_RUNG wire#w1
   // the same network as SCL:
   #_w1 := "DB16000_OPC_UA_TRIGGER_ALARM".CLIENT.U1_STA3_COAXIAL.TRIGGERS.START_CAM_NOZZLE_ANALISIS AND NOT "DB16000_OPC_UA_TRIGGER_ALARM".CLIENT.U1_STA3_COAXIAL.TRIGGERS.START_CAM_NOZZLE_ANALISIS_P;   // rising edge
   "DB16000_OPC_UA_TRIGGER_ALARM".CLIENT.U1_STA3_COAXIAL.TRIGGERS.START_CAM_NOZZLE_ANALISIS_P := "DB16000_OPC_UA_TRIGGER_ALARM".CLIENT.U1_STA3_COAXIAL.TRIGGERS.START_CAM_NOZZLE_ANALISIS;
   IF "M_DUMMY_OFF" THEN
       "DB16215_METHODCALL_U01_STA3_CAM_NOZZLE_ANALISIS_TRIGGER"(REQ := #_w1,   // OPC_UA_MethodCall_C
                               MaintainSession := false,
                               ServerEndpointUrl := "DB16102_U01_STA3_CAM_CLIENT_CONFIGURATION".Connection.ServerEndpointUrl,
                               SessionConnectInfo := "DB16102_U01_STA3_CAM_CLIENT_CONFIGURATION".Connection.ConnectInfo,
                               NamespaceUrisCount := "DB16102_U01_STA3_CAM_CLIENT_CONFIGURATION".Namespaces.NamespaceCount,
                               MethodHdlCount := "DB16102_U01_STA3_CAM_CLIENT_CONFIGURATION".MethodLists.U1_STA3_CAM_Analysis.MethodCount,
                               MethodHdl := "DB16102_U01_STA3_CAM_CLIENT_CONFIGURATION".MethodLists.U1_STA3_CAM_Analysis.MethodHdls[0],
                               NamespaceUris := "DB16102_U01_STA3_CAM_CLIENT_CONFIGURATION".Namespaces.NamespaceURIs,
                               NamespaceStatusList := "DB16102_U01_STA3_CAM_CLIENT_CONFIGURATION".Namespaces.NamespaceStatusList,
                               NamespaceIndexes := "DB16102_U01_STA3_CAM_CLIENT_CONFIGURATION".Namespaces.ServerNamespaceIndexes,
                               ObjectNodeIDs := "DB16102_U01_STA3_CAM_CLIENT_CONFIGURATION".MethodLists.U1_STA3_CAM_Analysis.ObjectNodes,
                               MethodNodeIDs := "DB16102_U01_STA3_CAM_CLIENT_CONFIGURATION".MethodLists.U1_STA3_CAM_Analysis.MethodNodes,
                               MethodHdls := "DB16102_U01_STA3_CAM_CLIENT_CONFIGURATION".MethodLists.U1_STA3_CAM_Analysis.MethodHdls,
                               StatusList := "DB16002_U01_STA3_COAXIAL_CLIENT_INTERFACE".U1_STA3_CAM_Analysis.MethodStatusList,
                               MethodResult := "DB16002_U01_STA3_COAXIAL_CLIENT_INTERFACE".U1_STA3_CAM_Analysis.MethodResultList[0],
                               OutputArguments := "DB16002_U01_STA3_COAXIAL_CLIENT_INTERFACE".U1_STA3_CAM_Analysis."Analyze nozzle".Outputs);
   END_IF;
END_REGION

REGION Network 19: UNIT 01 STATION 3 COAXIAL CAMERA START JET ANALISIS TRIGGER CALL
   // CAMBIAR POR EL METODO CORRECTO
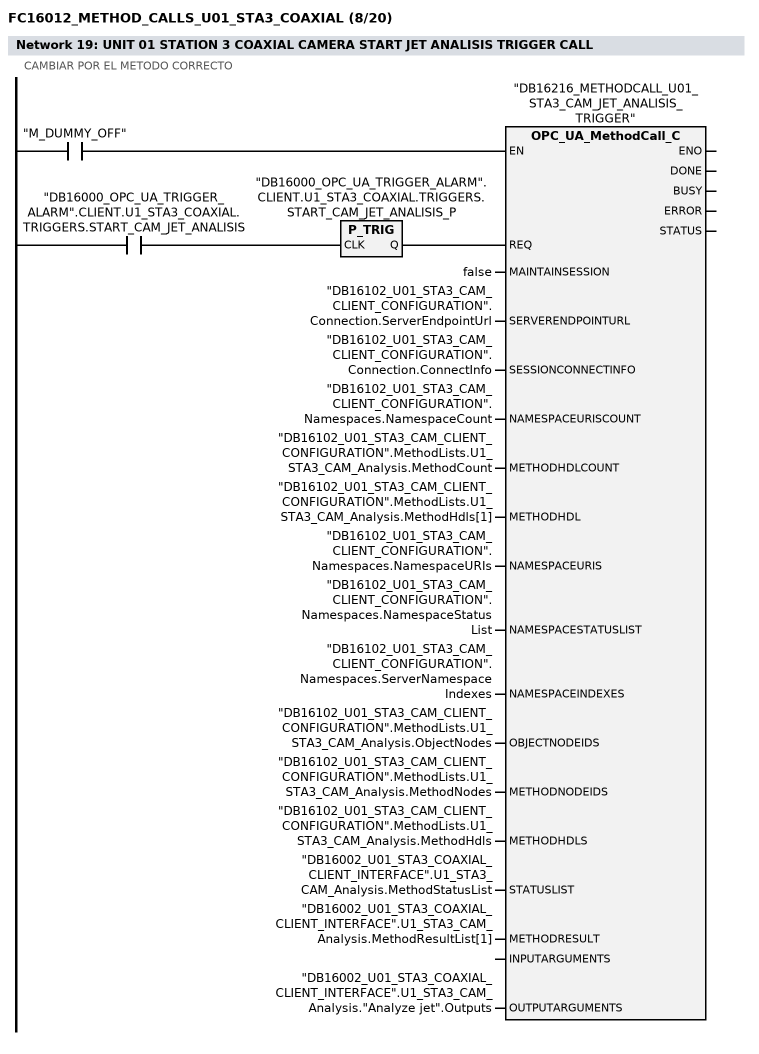
   RUNG wire#powerrail
      Contact( "M_DUMMY_OFF" )
      "DB16216_METHODCALL_U01_STA3_CAM_JET_ANALISIS_TRIGGER".OPC_UA_MethodCall_C(REQ := wire#w1, MaintainSession := false, ServerEndpointUrl := "DB16102_U01_STA3_CAM_CLIENT_CONFIGURATION".Connection.ServerEndpointUrl, SessionConnectInfo := "DB16102_U01_STA3_CAM_CLIENT_CONFIGURATION".Connection.ConnectInfo, NamespaceUrisCount := "DB16102_U01_STA3_CAM_CLIENT_CONFIGURATION".Namespaces.NamespaceCount, MethodHdlCount := "DB16102_U01_STA3_CAM_CLIENT_CONFIGURATION".MethodLists.U1_STA3_CAM_Analysis.MethodCount, MethodHdl := "DB16102_U01_STA3_CAM_CLIENT_CONFIGURATION".MethodLists.U1_STA3_CAM_Analysis.MethodHdls[1], NamespaceUris := "DB16102_U01_STA3_CAM_CLIENT_CONFIGURATION".Namespaces.NamespaceURIs, NamespaceStatusList := "DB16102_U01_STA3_CAM_CLIENT_CONFIGURATION".Namespaces.NamespaceStatusList, NamespaceIndexes := "DB16102_U01_STA3_CAM_CLIENT_CONFIGURATION".Namespaces.ServerNamespaceIndexes, ObjectNodeIDs := "DB16102_U01_STA3_CAM_CLIENT_CONFIGURATION".MethodLists.U1_STA3_CAM_Analysis.ObjectNodes, MethodNodeIDs := "DB16102_U01_STA3_CAM_CLIENT_CONFIGURATION".MethodLists.U1_STA3_CAM_Analysis.MethodNodes, MethodHdls := "DB16102_U01_STA3_CAM_CLIENT_CONFIGURATION".MethodLists.U1_STA3_CAM_Analysis.MethodHdls, StatusList := "DB16002_U01_STA3_COAXIAL_CLIENT_INTERFACE".U1_STA3_CAM_Analysis.MethodStatusList, MethodResult := "DB16002_U01_STA3_COAXIAL_CLIENT_INTERFACE".U1_STA3_CAM_Analysis.MethodResultList[1], InputArguments :=, OutputArguments := "DB16002_U01_STA3_COAXIAL_CLIENT_INTERFACE".U1_STA3_CAM_Analysis."Analyze jet".Outputs, Done =>, Busy =>, Error =>, Status =>)
   END_RUNG
   RUNG wire#powerrail
      Contact( "DB16000_OPC_UA_TRIGGER_ALARM".CLIENT.U1_STA3_COAXIAL.TRIGGERS.START_CAM_JET_ANALISIS )
      P_Trig( "DB16000_OPC_UA_TRIGGER_ALARM".CLIENT.U1_STA3_COAXIAL.TRIGGERS.START_CAM_JET_ANALISIS_P )
   END_RUNG wire#w1
   // the same network as SCL:
   #_w1 := "DB16000_OPC_UA_TRIGGER_ALARM".CLIENT.U1_STA3_COAXIAL.TRIGGERS.START_CAM_JET_ANALISIS AND NOT "DB16000_OPC_UA_TRIGGER_ALARM".CLIENT.U1_STA3_COAXIAL.TRIGGERS.START_CAM_JET_ANALISIS_P;   // rising edge
   "DB16000_OPC_UA_TRIGGER_ALARM".CLIENT.U1_STA3_COAXIAL.TRIGGERS.START_CAM_JET_ANALISIS_P := "DB16000_OPC_UA_TRIGGER_ALARM".CLIENT.U1_STA3_COAXIAL.TRIGGERS.START_CAM_JET_ANALISIS;
   IF "M_DUMMY_OFF" THEN
       "DB16216_METHODCALL_U01_STA3_CAM_JET_ANALISIS_TRIGGER"(REQ := #_w1,   // OPC_UA_MethodCall_C
                               MaintainSession := false,
                               ServerEndpointUrl := "DB16102_U01_STA3_CAM_CLIENT_CONFIGURATION".Connection.ServerEndpointUrl,
                               SessionConnectInfo := "DB16102_U01_STA3_CAM_CLIENT_CONFIGURATION".Connection.ConnectInfo,
                               NamespaceUrisCount := "DB16102_U01_STA3_CAM_CLIENT_CONFIGURATION".Namespaces.NamespaceCount,
                               MethodHdlCount := "DB16102_U01_STA3_CAM_CLIENT_CONFIGURATION".MethodLists.U1_STA3_CAM_Analysis.MethodCount,
                               MethodHdl := "DB16102_U01_STA3_CAM_CLIENT_CONFIGURATION".MethodLists.U1_STA3_CAM_Analysis.MethodHdls[1],
                               NamespaceUris := "DB16102_U01_STA3_CAM_CLIENT_CONFIGURATION".Namespaces.NamespaceURIs,
                               NamespaceStatusList := "DB16102_U01_STA3_CAM_CLIENT_CONFIGURATION".Namespaces.NamespaceStatusList,
                               NamespaceIndexes := "DB16102_U01_STA3_CAM_CLIENT_CONFIGURATION".Namespaces.ServerNamespaceIndexes,
                               ObjectNodeIDs := "DB16102_U01_STA3_CAM_CLIENT_CONFIGURATION".MethodLists.U1_STA3_CAM_Analysis.ObjectNodes,
                               MethodNodeIDs := "DB16102_U01_STA3_CAM_CLIENT_CONFIGURATION".MethodLists.U1_STA3_CAM_Analysis.MethodNodes,
                               MethodHdls := "DB16102_U01_STA3_CAM_CLIENT_CONFIGURATION".MethodLists.U1_STA3_CAM_Analysis.MethodHdls,
                               StatusList := "DB16002_U01_STA3_COAXIAL_CLIENT_INTERFACE".U1_STA3_CAM_Analysis.MethodStatusList,
                               MethodResult := "DB16002_U01_STA3_COAXIAL_CLIENT_INTERFACE".U1_STA3_CAM_Analysis.MethodResultList[1],
                               OutputArguments := "DB16002_U01_STA3_COAXIAL_CLIENT_INTERFACE".U1_STA3_CAM_Analysis."Analyze jet".Outputs);
   END_IF;
END_REGION

REGION Network 20: UNIT 01 STATION 3 COAXIAL CAMERA START CLADDING ANALISIS TRIGGER CALL
   // CAMBIAR POR EL METODO CORRECTO
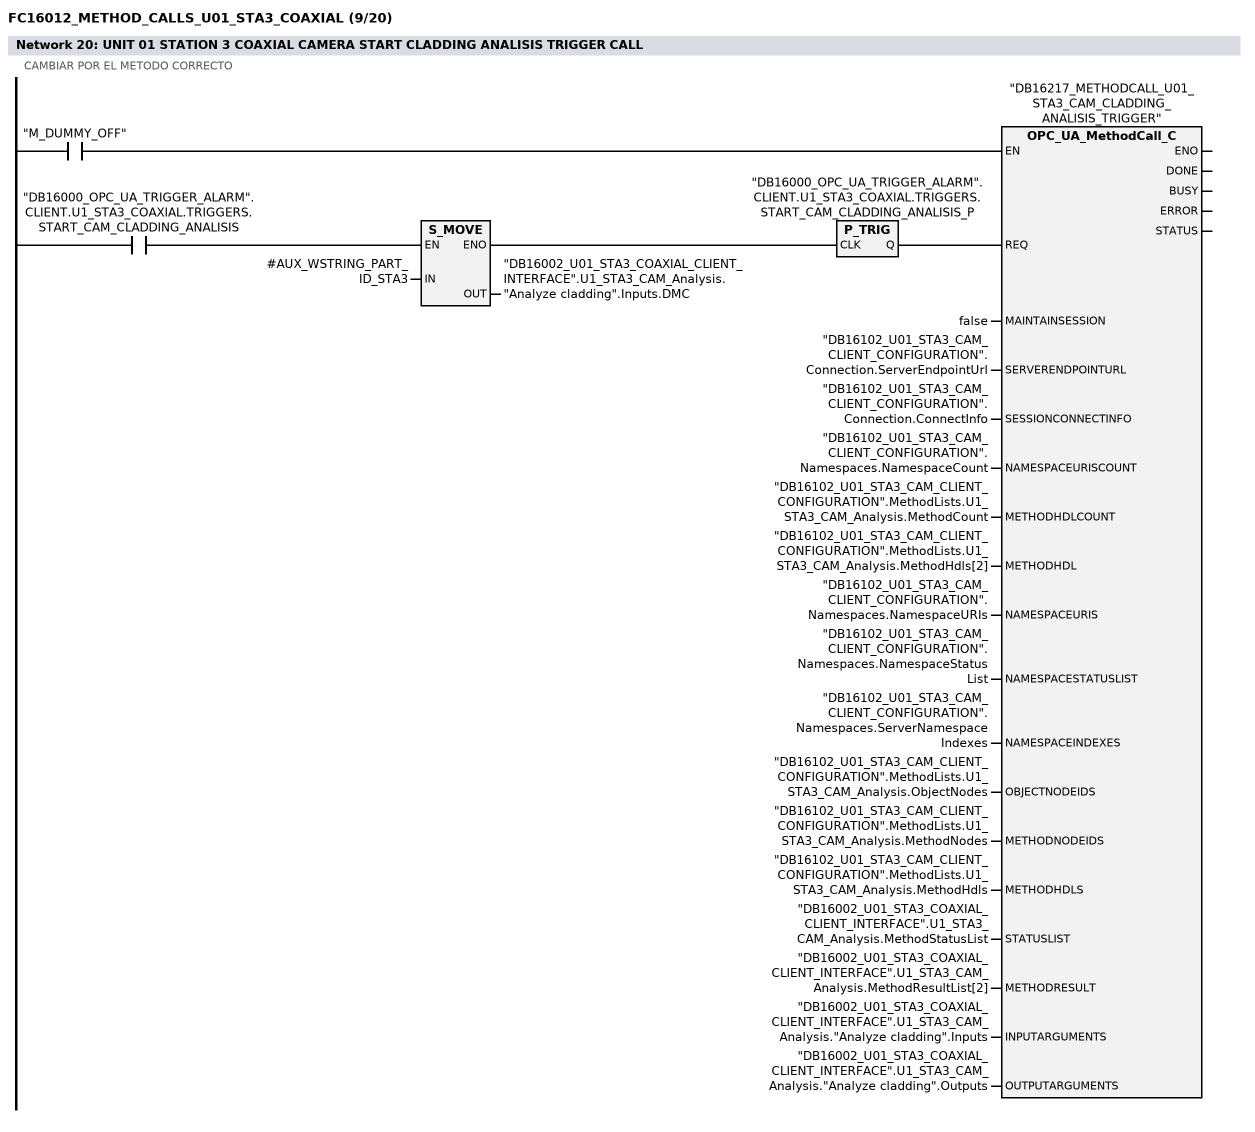
   RUNG wire#powerrail
      Contact( "M_DUMMY_OFF" )
      "DB16217_METHODCALL_U01_STA3_CAM_CLADDING_ANALISIS_TRIGGER".OPC_UA_MethodCall_C(REQ := wire#w1, MaintainSession := false, ServerEndpointUrl := "DB16102_U01_STA3_CAM_CLIENT_CONFIGURATION".Connection.ServerEndpointUrl, SessionConnectInfo := "DB16102_U01_STA3_CAM_CLIENT_CONFIGURATION".Connection.ConnectInfo, NamespaceUrisCount := "DB16102_U01_STA3_CAM_CLIENT_CONFIGURATION".Namespaces.NamespaceCount, MethodHdlCount := "DB16102_U01_STA3_CAM_CLIENT_CONFIGURATION".MethodLists.U1_STA3_CAM_Analysis.MethodCount, MethodHdl := "DB16102_U01_STA3_CAM_CLIENT_CONFIGURATION".MethodLists.U1_STA3_CAM_Analysis.MethodHdls[2], NamespaceUris := "DB16102_U01_STA3_CAM_CLIENT_CONFIGURATION".Namespaces.NamespaceURIs, NamespaceStatusList := "DB16102_U01_STA3_CAM_CLIENT_CONFIGURATION".Namespaces.NamespaceStatusList, NamespaceIndexes := "DB16102_U01_STA3_CAM_CLIENT_CONFIGURATION".Namespaces.ServerNamespaceIndexes, ObjectNodeIDs := "DB16102_U01_STA3_CAM_CLIENT_CONFIGURATION".MethodLists.U1_STA3_CAM_Analysis.ObjectNodes, MethodNodeIDs := "DB16102_U01_STA3_CAM_CLIENT_CONFIGURATION".MethodLists.U1_STA3_CAM_Analysis.MethodNodes, MethodHdls := "DB16102_U01_STA3_CAM_CLIENT_CONFIGURATION".MethodLists.U1_STA3_CAM_Analysis.MethodHdls, StatusList := "DB16002_U01_STA3_COAXIAL_CLIENT_INTERFACE".U1_STA3_CAM_Analysis.MethodStatusList, MethodResult := "DB16002_U01_STA3_COAXIAL_CLIENT_INTERFACE".U1_STA3_CAM_Analysis.MethodResultList[2], InputArguments := "DB16002_U01_STA3_COAXIAL_CLIENT_INTERFACE".U1_STA3_CAM_Analysis."Analyze cladding".Inputs, OutputArguments := "DB16002_U01_STA3_COAXIAL_CLIENT_INTERFACE".U1_STA3_CAM_Analysis."Analyze cladding".Outputs, Done =>, Busy =>, Error =>, Status =>)
   END_RUNG
   RUNG wire#powerrail
      Contact( "DB16000_OPC_UA_TRIGGER_ALARM".CLIENT.U1_STA3_COAXIAL.TRIGGERS.START_CAM_CLADDING_ANALISIS )
      S_Move(in := #AUX_WSTRING_PART_ID_STA3, out => "DB16002_U01_STA3_COAXIAL_CLIENT_INTERFACE".U1_STA3_CAM_Analysis."Analyze cladding".Inputs.DMC)
      P_Trig( "DB16000_OPC_UA_TRIGGER_ALARM".CLIENT.U1_STA3_COAXIAL.TRIGGERS.START_CAM_CLADDING_ANALISIS_P )
   END_RUNG wire#w1
   // the same network as SCL:
   IF "DB16000_OPC_UA_TRIGGER_ALARM".CLIENT.U1_STA3_COAXIAL.TRIGGERS.START_CAM_CLADDING_ANALISIS THEN
       "DB16002_U01_STA3_COAXIAL_CLIENT_INTERFACE".U1_STA3_CAM_Analysis."Analyze cladding".Inputs.DMC := #AUX_WSTRING_PART_ID_STA3;
   END_IF;
   #_w1 := "DB16000_OPC_UA_TRIGGER_ALARM".CLIENT.U1_STA3_COAXIAL.TRIGGERS.START_CAM_CLADDING_ANALISIS AND NOT "DB16000_OPC_UA_TRIGGER_ALARM".CLIENT.U1_STA3_COAXIAL.TRIGGERS.START_CAM_CLADDING_ANALISIS_P;   // rising edge
   "DB16000_OPC_UA_TRIGGER_ALARM".CLIENT.U1_STA3_COAXIAL.TRIGGERS.START_CAM_CLADDING_ANALISIS_P := "DB16000_OPC_UA_TRIGGER_ALARM".CLIENT.U1_STA3_COAXIAL.TRIGGERS.START_CAM_CLADDING_ANALISIS;
   IF "M_DUMMY_OFF" THEN
       "DB16217_METHODCALL_U01_STA3_CAM_CLADDING_ANALISIS_TRIGGER"(REQ := #_w1,   // OPC_UA_MethodCall_C
                               MaintainSession := false,
                               ServerEndpointUrl := "DB16102_U01_STA3_CAM_CLIENT_CONFIGURATION".Connection.ServerEndpointUrl,
                               SessionConnectInfo := "DB16102_U01_STA3_CAM_CLIENT_CONFIGURATION".Connection.ConnectInfo,
                               NamespaceUrisCount := "DB16102_U01_STA3_CAM_CLIENT_CONFIGURATION".Namespaces.NamespaceCount,
                               MethodHdlCount := "DB16102_U01_STA3_CAM_CLIENT_CONFIGURATION".MethodLists.U1_STA3_CAM_Analysis.MethodCount,
                               MethodHdl := "DB16102_U01_STA3_CAM_CLIENT_CONFIGURATION".MethodLists.U1_STA3_CAM_Analysis.MethodHdls[2],
                               NamespaceUris := "DB16102_U01_STA3_CAM_CLIENT_CONFIGURATION".Namespaces.NamespaceURIs,
                               NamespaceStatusList := "DB16102_U01_STA3_CAM_CLIENT_CONFIGURATION".Namespaces.NamespaceStatusList,
                               NamespaceIndexes := "DB16102_U01_STA3_CAM_CLIENT_CONFIGURATION".Namespaces.ServerNamespaceIndexes,
                               ObjectNodeIDs := "DB16102_U01_STA3_CAM_CLIENT_CONFIGURATION".MethodLists.U1_STA3_CAM_Analysis.ObjectNodes,
                               MethodNodeIDs := "DB16102_U01_STA3_CAM_CLIENT_CONFIGURATION".MethodLists.U1_STA3_CAM_Analysis.MethodNodes,
                               MethodHdls := "DB16102_U01_STA3_CAM_CLIENT_CONFIGURATION".MethodLists.U1_STA3_CAM_Analysis.MethodHdls,
                               StatusList := "DB16002_U01_STA3_COAXIAL_CLIENT_INTERFACE".U1_STA3_CAM_Analysis.MethodStatusList,
                               MethodResult := "DB16002_U01_STA3_COAXIAL_CLIENT_INTERFACE".U1_STA3_CAM_Analysis.MethodResultList[2],
                               InputArguments := "DB16002_U01_STA3_COAXIAL_CLIENT_INTERFACE".U1_STA3_CAM_Analysis."Analyze cladding".Inputs,
                               OutputArguments := "DB16002_U01_STA3_COAXIAL_CLIENT_INTERFACE".U1_STA3_CAM_Analysis."Analyze cladding".Outputs);
   END_IF;
END_REGION

REGION Network 21: UNIT 01 STATION 3 COAXIAL CAMERA STOP METHODS TRIGGER CALL
   // CAMBIAR POR EL METODO CORRECTO
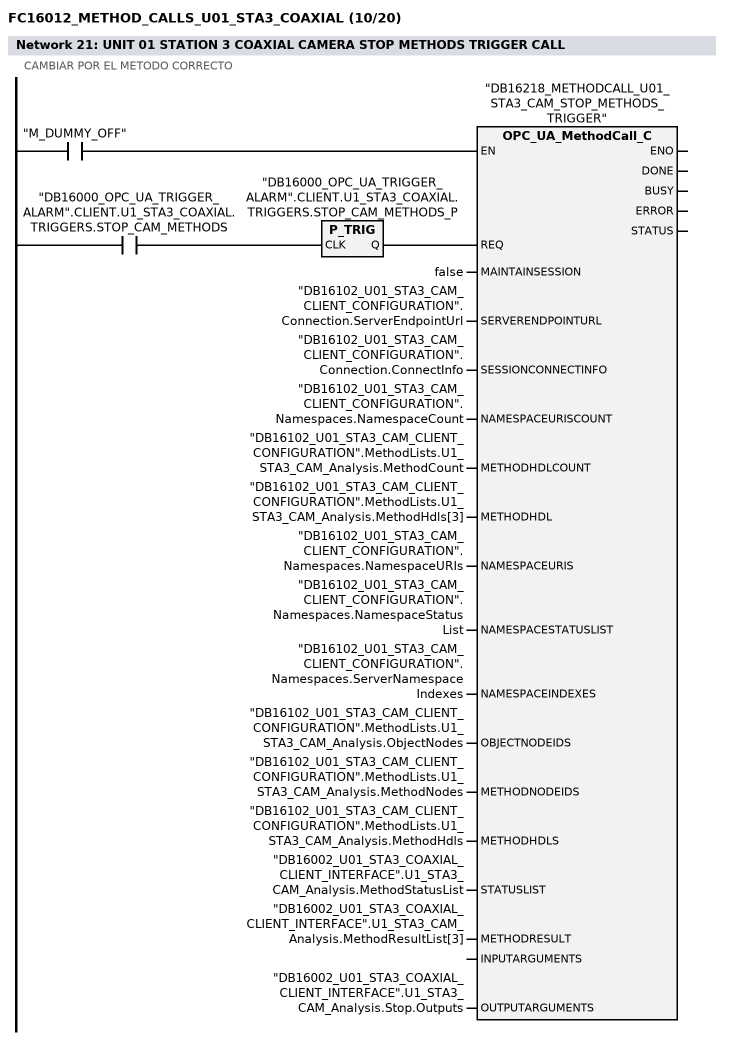
   RUNG wire#powerrail
      Contact( "M_DUMMY_OFF" )
      "DB16218_METHODCALL_U01_STA3_CAM_STOP_METHODS_TRIGGER".OPC_UA_MethodCall_C(REQ := wire#w1, MaintainSession := false, ServerEndpointUrl := "DB16102_U01_STA3_CAM_CLIENT_CONFIGURATION".Connection.ServerEndpointUrl, SessionConnectInfo := "DB16102_U01_STA3_CAM_CLIENT_CONFIGURATION".Connection.ConnectInfo, NamespaceUrisCount := "DB16102_U01_STA3_CAM_CLIENT_CONFIGURATION".Namespaces.NamespaceCount, MethodHdlCount := "DB16102_U01_STA3_CAM_CLIENT_CONFIGURATION".MethodLists.U1_STA3_CAM_Analysis.MethodCount, MethodHdl := "DB16102_U01_STA3_CAM_CLIENT_CONFIGURATION".MethodLists.U1_STA3_CAM_Analysis.MethodHdls[3], NamespaceUris := "DB16102_U01_STA3_CAM_CLIENT_CONFIGURATION".Namespaces.NamespaceURIs, NamespaceStatusList := "DB16102_U01_STA3_CAM_CLIENT_CONFIGURATION".Namespaces.NamespaceStatusList, NamespaceIndexes := "DB16102_U01_STA3_CAM_CLIENT_CONFIGURATION".Namespaces.ServerNamespaceIndexes, ObjectNodeIDs := "DB16102_U01_STA3_CAM_CLIENT_CONFIGURATION".MethodLists.U1_STA3_CAM_Analysis.ObjectNodes, MethodNodeIDs := "DB16102_U01_STA3_CAM_CLIENT_CONFIGURATION".MethodLists.U1_STA3_CAM_Analysis.MethodNodes, MethodHdls := "DB16102_U01_STA3_CAM_CLIENT_CONFIGURATION".MethodLists.U1_STA3_CAM_Analysis.MethodHdls, StatusList := "DB16002_U01_STA3_COAXIAL_CLIENT_INTERFACE".U1_STA3_CAM_Analysis.MethodStatusList, MethodResult := "DB16002_U01_STA3_COAXIAL_CLIENT_INTERFACE".U1_STA3_CAM_Analysis.MethodResultList[3], InputArguments :=, OutputArguments := "DB16002_U01_STA3_COAXIAL_CLIENT_INTERFACE".U1_STA3_CAM_Analysis.Stop.Outputs, Done =>, Busy =>, Error =>, Status =>)
   END_RUNG
   RUNG wire#powerrail
      Contact( "DB16000_OPC_UA_TRIGGER_ALARM".CLIENT.U1_STA3_COAXIAL.TRIGGERS.STOP_CAM_METHODS )
      P_Trig( "DB16000_OPC_UA_TRIGGER_ALARM".CLIENT.U1_STA3_COAXIAL.TRIGGERS.STOP_CAM_METHODS_P )
   END_RUNG wire#w1
   // the same network as SCL:
   #_w1 := "DB16000_OPC_UA_TRIGGER_ALARM".CLIENT.U1_STA3_COAXIAL.TRIGGERS.STOP_CAM_METHODS AND NOT "DB16000_OPC_UA_TRIGGER_ALARM".CLIENT.U1_STA3_COAXIAL.TRIGGERS.STOP_CAM_METHODS_P;   // rising edge
   "DB16000_OPC_UA_TRIGGER_ALARM".CLIENT.U1_STA3_COAXIAL.TRIGGERS.STOP_CAM_METHODS_P := "DB16000_OPC_UA_TRIGGER_ALARM".CLIENT.U1_STA3_COAXIAL.TRIGGERS.STOP_CAM_METHODS;
   IF "M_DUMMY_OFF" THEN
       "DB16218_METHODCALL_U01_STA3_CAM_STOP_METHODS_TRIGGER"(REQ := #_w1,   // OPC_UA_MethodCall_C
                               MaintainSession := false,
                               ServerEndpointUrl := "DB16102_U01_STA3_CAM_CLIENT_CONFIGURATION".Connection.ServerEndpointUrl,
                               SessionConnectInfo := "DB16102_U01_STA3_CAM_CLIENT_CONFIGURATION".Connection.ConnectInfo,
                               NamespaceUrisCount := "DB16102_U01_STA3_CAM_CLIENT_CONFIGURATION".Namespaces.NamespaceCount,
                               MethodHdlCount := "DB16102_U01_STA3_CAM_CLIENT_CONFIGURATION".MethodLists.U1_STA3_CAM_Analysis.MethodCount,
                               MethodHdl := "DB16102_U01_STA3_CAM_CLIENT_CONFIGURATION".MethodLists.U1_STA3_CAM_Analysis.MethodHdls[3],
                               NamespaceUris := "DB16102_U01_STA3_CAM_CLIENT_CONFIGURATION".Namespaces.NamespaceURIs,
                               NamespaceStatusList := "DB16102_U01_STA3_CAM_CLIENT_CONFIGURATION".Namespaces.NamespaceStatusList,
                               NamespaceIndexes := "DB16102_U01_STA3_CAM_CLIENT_CONFIGURATION".Namespaces.ServerNamespaceIndexes,
                               ObjectNodeIDs := "DB16102_U01_STA3_CAM_CLIENT_CONFIGURATION".MethodLists.U1_STA3_CAM_Analysis.ObjectNodes,
                               MethodNodeIDs := "DB16102_U01_STA3_CAM_CLIENT_CONFIGURATION".MethodLists.U1_STA3_CAM_Analysis.MethodNodes,
                               MethodHdls := "DB16102_U01_STA3_CAM_CLIENT_CONFIGURATION".MethodLists.U1_STA3_CAM_Analysis.MethodHdls,
                               StatusList := "DB16002_U01_STA3_COAXIAL_CLIENT_INTERFACE".U1_STA3_CAM_Analysis.MethodStatusList,
                               MethodResult := "DB16002_U01_STA3_COAXIAL_CLIENT_INTERFACE".U1_STA3_CAM_Analysis.MethodResultList[3],
                               OutputArguments := "DB16002_U01_STA3_COAXIAL_CLIENT_INTERFACE".U1_STA3_CAM_Analysis.Stop.Outputs);
   END_IF;
END_REGION

REGION Network 22: UNIT 01 STATION 3 COAXIAL CAMERA RESET PC TRIGGER CALL
   // CAMBIAR POR EL METODO CORRECTO
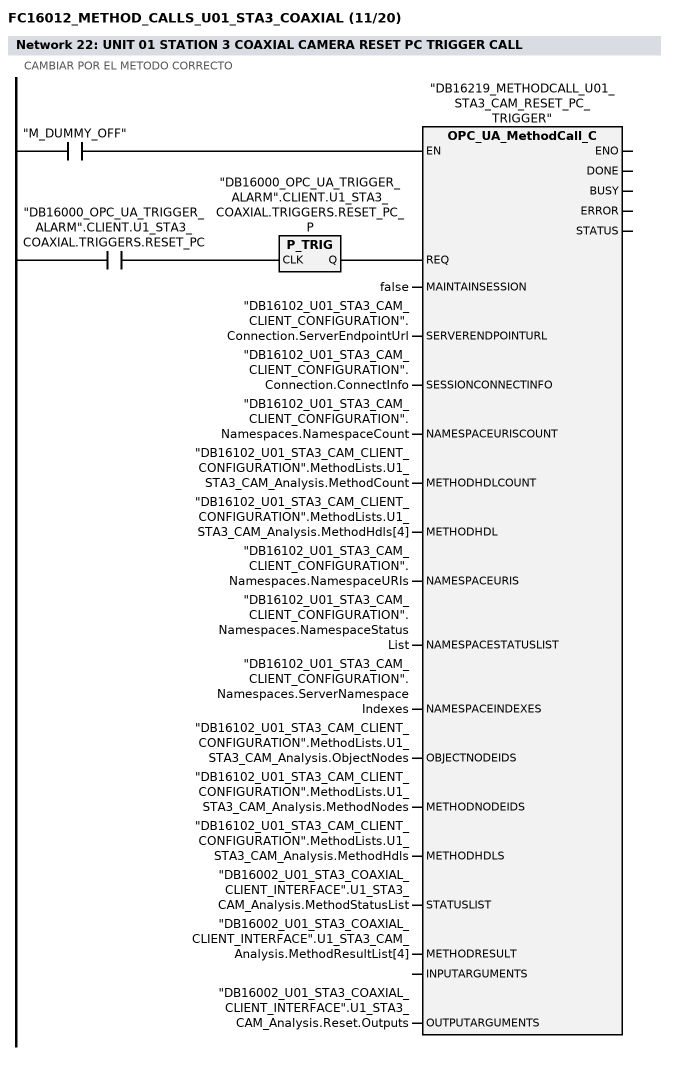
   RUNG wire#powerrail
      Contact( "M_DUMMY_OFF" )
      "DB16219_METHODCALL_U01_STA3_CAM_RESET_PC_TRIGGER".OPC_UA_MethodCall_C(REQ := wire#w1, MaintainSession := false, ServerEndpointUrl := "DB16102_U01_STA3_CAM_CLIENT_CONFIGURATION".Connection.ServerEndpointUrl, SessionConnectInfo := "DB16102_U01_STA3_CAM_CLIENT_CONFIGURATION".Connection.ConnectInfo, NamespaceUrisCount := "DB16102_U01_STA3_CAM_CLIENT_CONFIGURATION".Namespaces.NamespaceCount, MethodHdlCount := "DB16102_U01_STA3_CAM_CLIENT_CONFIGURATION".MethodLists.U1_STA3_CAM_Analysis.MethodCount, MethodHdl := "DB16102_U01_STA3_CAM_CLIENT_CONFIGURATION".MethodLists.U1_STA3_CAM_Analysis.MethodHdls[4], NamespaceUris := "DB16102_U01_STA3_CAM_CLIENT_CONFIGURATION".Namespaces.NamespaceURIs, NamespaceStatusList := "DB16102_U01_STA3_CAM_CLIENT_CONFIGURATION".Namespaces.NamespaceStatusList, NamespaceIndexes := "DB16102_U01_STA3_CAM_CLIENT_CONFIGURATION".Namespaces.ServerNamespaceIndexes, ObjectNodeIDs := "DB16102_U01_STA3_CAM_CLIENT_CONFIGURATION".MethodLists.U1_STA3_CAM_Analysis.ObjectNodes, MethodNodeIDs := "DB16102_U01_STA3_CAM_CLIENT_CONFIGURATION".MethodLists.U1_STA3_CAM_Analysis.MethodNodes, MethodHdls := "DB16102_U01_STA3_CAM_CLIENT_CONFIGURATION".MethodLists.U1_STA3_CAM_Analysis.MethodHdls, StatusList := "DB16002_U01_STA3_COAXIAL_CLIENT_INTERFACE".U1_STA3_CAM_Analysis.MethodStatusList, MethodResult := "DB16002_U01_STA3_COAXIAL_CLIENT_INTERFACE".U1_STA3_CAM_Analysis.MethodResultList[4], InputArguments :=, OutputArguments := "DB16002_U01_STA3_COAXIAL_CLIENT_INTERFACE".U1_STA3_CAM_Analysis.Reset.Outputs, Done =>, Busy =>, Error =>, Status =>)
   END_RUNG
   RUNG wire#powerrail
      Contact( "DB16000_OPC_UA_TRIGGER_ALARM".CLIENT.U1_STA3_COAXIAL.TRIGGERS.RESET_PC )
      P_Trig( "DB16000_OPC_UA_TRIGGER_ALARM".CLIENT.U1_STA3_COAXIAL.TRIGGERS.RESET_PC_P )
   END_RUNG wire#w1
   // the same network as SCL:
   #_w1 := "DB16000_OPC_UA_TRIGGER_ALARM".CLIENT.U1_STA3_COAXIAL.TRIGGERS.RESET_PC AND NOT "DB16000_OPC_UA_TRIGGER_ALARM".CLIENT.U1_STA3_COAXIAL.TRIGGERS.RESET_PC_P;   // rising edge
   "DB16000_OPC_UA_TRIGGER_ALARM".CLIENT.U1_STA3_COAXIAL.TRIGGERS.RESET_PC_P := "DB16000_OPC_UA_TRIGGER_ALARM".CLIENT.U1_STA3_COAXIAL.TRIGGERS.RESET_PC;
   IF "M_DUMMY_OFF" THEN
       "DB16219_METHODCALL_U01_STA3_CAM_RESET_PC_TRIGGER"(REQ := #_w1,   // OPC_UA_MethodCall_C
                               MaintainSession := false,
                               ServerEndpointUrl := "DB16102_U01_STA3_CAM_CLIENT_CONFIGURATION".Connection.ServerEndpointUrl,
                               SessionConnectInfo := "DB16102_U01_STA3_CAM_CLIENT_CONFIGURATION".Connection.ConnectInfo,
                               NamespaceUrisCount := "DB16102_U01_STA3_CAM_CLIENT_CONFIGURATION".Namespaces.NamespaceCount,
                               MethodHdlCount := "DB16102_U01_STA3_CAM_CLIENT_CONFIGURATION".MethodLists.U1_STA3_CAM_Analysis.MethodCount,
                               MethodHdl := "DB16102_U01_STA3_CAM_CLIENT_CONFIGURATION".MethodLists.U1_STA3_CAM_Analysis.MethodHdls[4],
                               NamespaceUris := "DB16102_U01_STA3_CAM_CLIENT_CONFIGURATION".Namespaces.NamespaceURIs,
                               NamespaceStatusList := "DB16102_U01_STA3_CAM_CLIENT_CONFIGURATION".Namespaces.NamespaceStatusList,
                               NamespaceIndexes := "DB16102_U01_STA3_CAM_CLIENT_CONFIGURATION".Namespaces.ServerNamespaceIndexes,
                               ObjectNodeIDs := "DB16102_U01_STA3_CAM_CLIENT_CONFIGURATION".MethodLists.U1_STA3_CAM_Analysis.ObjectNodes,
                               MethodNodeIDs := "DB16102_U01_STA3_CAM_CLIENT_CONFIGURATION".MethodLists.U1_STA3_CAM_Analysis.MethodNodes,
                               MethodHdls := "DB16102_U01_STA3_CAM_CLIENT_CONFIGURATION".MethodLists.U1_STA3_CAM_Analysis.MethodHdls,
                               StatusList := "DB16002_U01_STA3_COAXIAL_CLIENT_INTERFACE".U1_STA3_CAM_Analysis.MethodStatusList,
                               MethodResult := "DB16002_U01_STA3_COAXIAL_CLIENT_INTERFACE".U1_STA3_CAM_Analysis.MethodResultList[4],
                               OutputArguments := "DB16002_U01_STA3_COAXIAL_CLIENT_INTERFACE".U1_STA3_CAM_Analysis.Reset.Outputs);
   END_IF;
END_REGION

REGION Network 23: UNIT 01 STATION 3 COAXIAL CAMERA READ VARIABLES TRIGGER CALL
   // CAMBIAR POR EL METODO CORRECTO
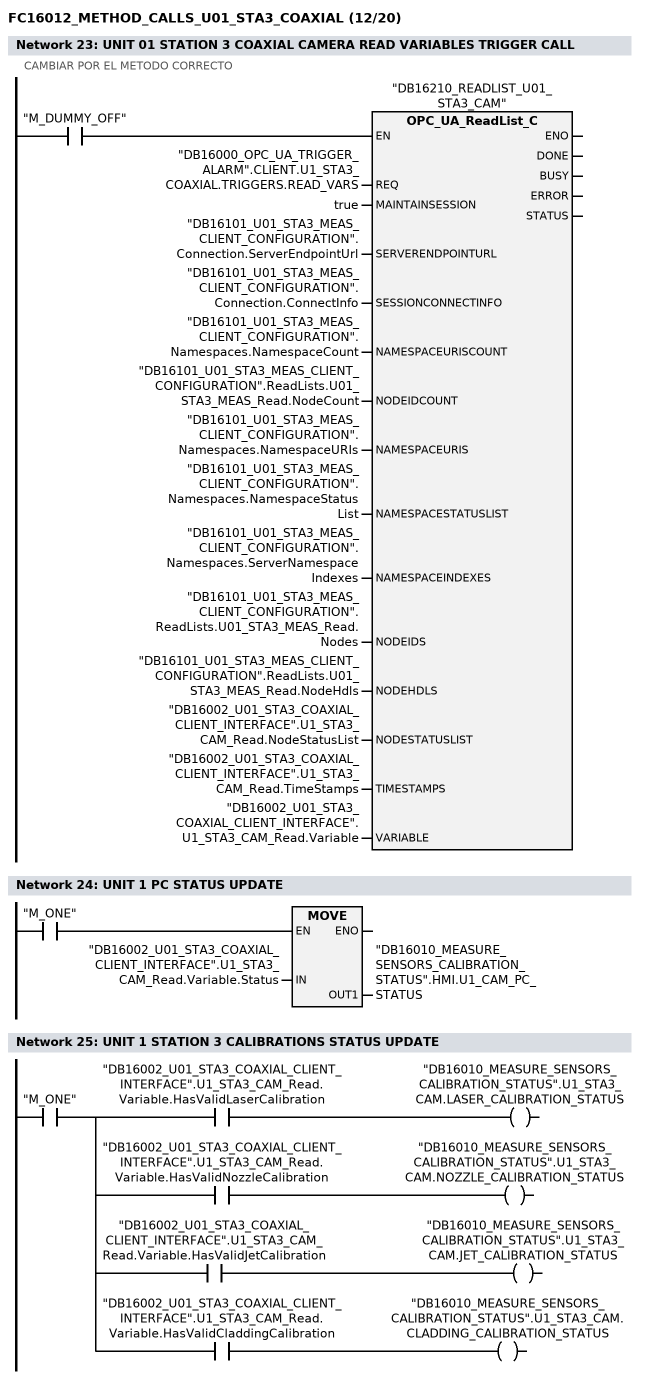
   RUNG wire#powerrail
      Contact( "M_DUMMY_OFF" )
      "DB16210_READLIST_U01_STA3_CAM".OPC_UA_ReadList_C(REQ := "DB16000_OPC_UA_TRIGGER_ALARM".CLIENT.U1_STA3_COAXIAL.TRIGGERS.READ_VARS, MaintainSession := true, ServerEndpointUrl := "DB16101_U01_STA3_MEAS_CLIENT_CONFIGURATION".Connection.ServerEndpointUrl, SessionConnectInfo := "DB16101_U01_STA3_MEAS_CLIENT_CONFIGURATION".Connection.ConnectInfo, NamespaceUrisCount := "DB16101_U01_STA3_MEAS_CLIENT_CONFIGURATION".Namespaces.NamespaceCount, NodeIDCount := "DB16101_U01_STA3_MEAS_CLIENT_CONFIGURATION".ReadLists.U01_STA3_MEAS_Read.NodeCount, NamespaceUris := "DB16101_U01_STA3_MEAS_CLIENT_CONFIGURATION".Namespaces.NamespaceURIs, NamespaceStatusList := "DB16101_U01_STA3_MEAS_CLIENT_CONFIGURATION".Namespaces.NamespaceStatusList, NamespaceIndexes := "DB16101_U01_STA3_MEAS_CLIENT_CONFIGURATION".Namespaces.ServerNamespaceIndexes, NodeIDs := "DB16101_U01_STA3_MEAS_CLIENT_CONFIGURATION".ReadLists.U01_STA3_MEAS_Read.Nodes, NodeHdls := "DB16101_U01_STA3_MEAS_CLIENT_CONFIGURATION".ReadLists.U01_STA3_MEAS_Read.NodeHdls, NodeStatusList := "DB16002_U01_STA3_COAXIAL_CLIENT_INTERFACE".U1_STA3_CAM_Read.NodeStatusList, Timestamps := "DB16002_U01_STA3_COAXIAL_CLIENT_INTERFACE".U1_STA3_CAM_Read.TimeStamps, Variable := "DB16002_U01_STA3_COAXIAL_CLIENT_INTERFACE".U1_STA3_CAM_Read.Variable, Done =>, Busy =>, Error =>, Status =>)
   END_RUNG
   // the same network as SCL:
   IF "M_DUMMY_OFF" THEN
       "DB16210_READLIST_U01_STA3_CAM"(REQ := "DB16000_OPC_UA_TRIGGER_ALARM".CLIENT.U1_STA3_COAXIAL.TRIGGERS.READ_VARS,   // OPC_UA_ReadList_C
                               MaintainSession := true,
                               ServerEndpointUrl := "DB16101_U01_STA3_MEAS_CLIENT_CONFIGURATION".Connection.ServerEndpointUrl,
                               SessionConnectInfo := "DB16101_U01_STA3_MEAS_CLIENT_CONFIGURATION".Connection.ConnectInfo,
                               NamespaceUrisCount := "DB16101_U01_STA3_MEAS_CLIENT_CONFIGURATION".Namespaces.NamespaceCount,
                               NodeIDCount := "DB16101_U01_STA3_MEAS_CLIENT_CONFIGURATION".ReadLists.U01_STA3_MEAS_Read.NodeCount,
                               NamespaceUris := "DB16101_U01_STA3_MEAS_CLIENT_CONFIGURATION".Namespaces.NamespaceURIs,
                               NamespaceStatusList := "DB16101_U01_STA3_MEAS_CLIENT_CONFIGURATION".Namespaces.NamespaceStatusList,
                               NamespaceIndexes := "DB16101_U01_STA3_MEAS_CLIENT_CONFIGURATION".Namespaces.ServerNamespaceIndexes,
                               NodeIDs := "DB16101_U01_STA3_MEAS_CLIENT_CONFIGURATION".ReadLists.U01_STA3_MEAS_Read.Nodes,
                               NodeHdls := "DB16101_U01_STA3_MEAS_CLIENT_CONFIGURATION".ReadLists.U01_STA3_MEAS_Read.NodeHdls,
                               NodeStatusList := "DB16002_U01_STA3_COAXIAL_CLIENT_INTERFACE".U1_STA3_CAM_Read.NodeStatusList,
                               Timestamps := "DB16002_U01_STA3_COAXIAL_CLIENT_INTERFACE".U1_STA3_CAM_Read.TimeStamps,
                               Variable := "DB16002_U01_STA3_COAXIAL_CLIENT_INTERFACE".U1_STA3_CAM_Read.Variable);
   END_IF;
END_REGION

REGION Network 24: UNIT 1 PC STATUS UPDATE
   RUNG wire#powerrail
      Contact( "M_ONE" )
      Move(in := "DB16002_U01_STA3_COAXIAL_CLIENT_INTERFACE".U1_STA3_CAM_Read.Variable.Status, out1 => "DB16010_MEASURE_SENSORS_CALIBRATION_STATUS".HMI.U1_CAM_PC_STATUS)
   END_RUNG
   // the same network as SCL:
   IF "M_ONE" THEN
       "DB16010_MEASURE_SENSORS_CALIBRATION_STATUS".HMI.U1_CAM_PC_STATUS := "DB16002_U01_STA3_COAXIAL_CLIENT_INTERFACE".U1_STA3_CAM_Read.Variable.Status;
   END_IF;
END_REGION

REGION Network 25: UNIT 1 STATION 3 CALIBRATIONS STATUS UPDATE
   RUNG wire#powerrail
      Contact( "M_ONE" )
      wire#w1
      Contact( "DB16002_U01_STA3_COAXIAL_CLIENT_INTERFACE".U1_STA3_CAM_Read.Variable.HasValidLaserCalibration )
      Coil( "DB16010_MEASURE_SENSORS_CALIBRATION_STATUS".U1_STA3_CAM.LASER_CALIBRATION_STATUS )
   END_RUNG
   RUNG wire#w1
      Contact( "DB16002_U01_STA3_COAXIAL_CLIENT_INTERFACE".U1_STA3_CAM_Read.Variable.HasValidNozzleCalibration )
      Coil( "DB16010_MEASURE_SENSORS_CALIBRATION_STATUS".U1_STA3_CAM.NOZZLE_CALIBRATION_STATUS )
   END_RUNG
   RUNG wire#w1
      Contact( "DB16002_U01_STA3_COAXIAL_CLIENT_INTERFACE".U1_STA3_CAM_Read.Variable.HasValidJetCalibration )
      Coil( "DB16010_MEASURE_SENSORS_CALIBRATION_STATUS".U1_STA3_CAM.JET_CALIBRATION_STATUS )
   END_RUNG
   RUNG wire#w1
      Contact( "DB16002_U01_STA3_COAXIAL_CLIENT_INTERFACE".U1_STA3_CAM_Read.Variable.HasValidCladdingCalibration )
      Coil( "DB16010_MEASURE_SENSORS_CALIBRATION_STATUS".U1_STA3_CAM.CLADDING_CALIBRATION_STATUS )
   END_RUNG
   // the same network as SCL:
   "DB16010_MEASURE_SENSORS_CALIBRATION_STATUS".U1_STA3_CAM.LASER_CALIBRATION_STATUS := "M_ONE" AND "DB16002_U01_STA3_COAXIAL_CLIENT_INTERFACE".U1_STA3_CAM_Read.Variable.HasValidLaserCalibration;
   "DB16010_MEASURE_SENSORS_CALIBRATION_STATUS".U1_STA3_CAM.NOZZLE_CALIBRATION_STATUS := "M_ONE" AND "DB16002_U01_STA3_COAXIAL_CLIENT_INTERFACE".U1_STA3_CAM_Read.Variable.HasValidNozzleCalibration;
   "DB16010_MEASURE_SENSORS_CALIBRATION_STATUS".U1_STA3_CAM.JET_CALIBRATION_STATUS := "M_ONE" AND "DB16002_U01_STA3_COAXIAL_CLIENT_INTERFACE".U1_STA3_CAM_Read.Variable.HasValidJetCalibration;
   "DB16010_MEASURE_SENSORS_CALIBRATION_STATUS".U1_STA3_CAM.CLADDING_CALIBRATION_STATUS := "M_ONE" AND "DB16002_U01_STA3_COAXIAL_CLIENT_INTERFACE".U1_STA3_CAM_Read.Variable.HasValidCladdingCalibration;
END_REGION

REGION Network 26: UNIT 01 STATION 3 COAXIAL CAMERA START LASER CALIBRATION METHOD CONNECTION ALARM
   // CAMBIAR BIT DE ERROR DEL METODO CORRECTO
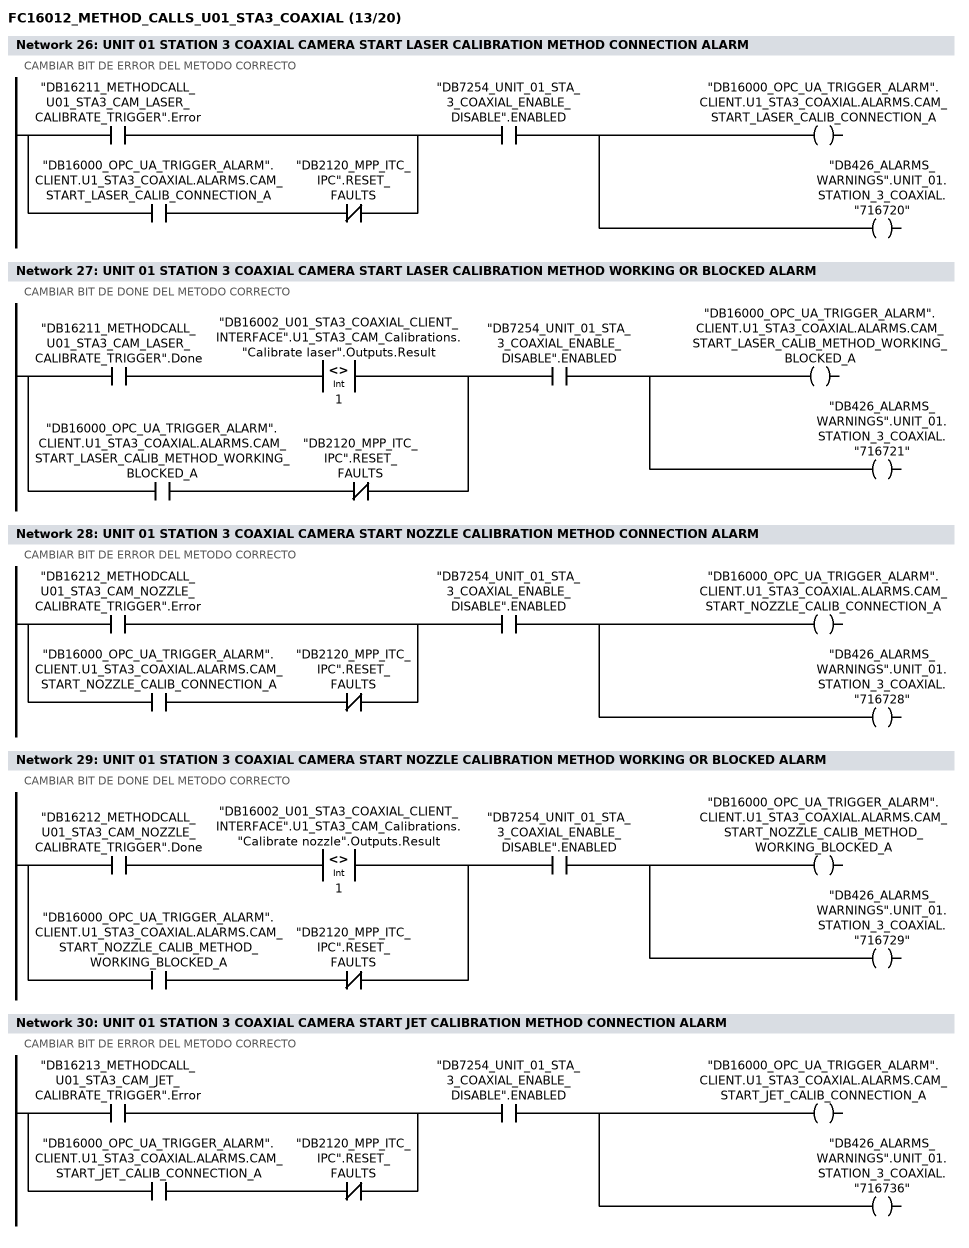
   RUNG wire#powerrail
      Contact( "DB16211_METHODCALL_U01_STA3_CAM_LASER_CALIBRATE_TRIGGER".Error )
      wire#w1
      Contact( "DB7254_UNIT_01_STA_3_COAXIAL_ENABLE_DISABLE".ENABLED )
      wire#w2
      Coil( "DB16000_OPC_UA_TRIGGER_ALARM".CLIENT.U1_STA3_COAXIAL.ALARMS.CAM_START_LASER_CALIB_CONNECTION_A )
   END_RUNG
   RUNG wire#powerrail
      Contact( "DB16000_OPC_UA_TRIGGER_ALARM".CLIENT.U1_STA3_COAXIAL.ALARMS.CAM_START_LASER_CALIB_CONNECTION_A )
      I_Contact( "DB2120_MPP_ITC_IPC".RESET_FAULTS )
   END_RUNG wire#w1
   RUNG wire#w2
      Coil( "DB426_ALARMS_WARNINGS".UNIT_01.STATION_3_COAXIAL."716720" )
   END_RUNG
   // the same network as SCL:
   "DB16000_OPC_UA_TRIGGER_ALARM".CLIENT.U1_STA3_COAXIAL.ALARMS.CAM_START_LASER_CALIB_CONNECTION_A := ("DB16211_METHODCALL_U01_STA3_CAM_LASER_CALIBRATE_TRIGGER".Error OR ("DB16000_OPC_UA_TRIGGER_ALARM".CLIENT.U1_STA3_COAXIAL.ALARMS.CAM_START_LASER_CALIB_CONNECTION_A AND NOT "DB2120_MPP_ITC_IPC".RESET_FAULTS)) AND "DB7254_UNIT_01_STA_3_COAXIAL_ENABLE_DISABLE".ENABLED;
   "DB426_ALARMS_WARNINGS".UNIT_01.STATION_3_COAXIAL."716720" := "DB16000_OPC_UA_TRIGGER_ALARM".CLIENT.U1_STA3_COAXIAL.ALARMS.CAM_START_LASER_CALIB_CONNECTION_A;
END_REGION

REGION Network 27: UNIT 01 STATION 3 COAXIAL CAMERA START LASER CALIBRATION METHOD WORKING OR BLOCKED ALARM
   // CAMBIAR BIT DE DONE DEL METODO CORRECTO
   RUNG wire#powerrail
      Contact( "DB16211_METHODCALL_U01_STA3_CAM_LASER_CALIBRATE_TRIGGER".Done )
      { S7_Templates := "SrcType := Int" } NE_Contact(in1 := "DB16002_U01_STA3_COAXIAL_CLIENT_INTERFACE".U1_STA3_CAM_Calibrations."Calibrate laser".Outputs.Result, in2 := 1)
      wire#w1
      Contact( "DB7254_UNIT_01_STA_3_COAXIAL_ENABLE_DISABLE".ENABLED )
      wire#w2
      Coil( "DB16000_OPC_UA_TRIGGER_ALARM".CLIENT.U1_STA3_COAXIAL.ALARMS.CAM_START_LASER_CALIB_METHOD_WORKING_BLOCKED_A )
   END_RUNG
   RUNG wire#powerrail
      Contact( "DB16000_OPC_UA_TRIGGER_ALARM".CLIENT.U1_STA3_COAXIAL.ALARMS.CAM_START_LASER_CALIB_METHOD_WORKING_BLOCKED_A )
      I_Contact( "DB2120_MPP_ITC_IPC".RESET_FAULTS )
   END_RUNG wire#w1
   RUNG wire#w2
      Coil( "DB426_ALARMS_WARNINGS".UNIT_01.STATION_3_COAXIAL."716721" )
   END_RUNG
   // the same network as SCL:
   "DB16000_OPC_UA_TRIGGER_ALARM".CLIENT.U1_STA3_COAXIAL.ALARMS.CAM_START_LASER_CALIB_METHOD_WORKING_BLOCKED_A := (("DB16211_METHODCALL_U01_STA3_CAM_LASER_CALIBRATE_TRIGGER".Done AND ("DB16002_U01_STA3_COAXIAL_CLIENT_INTERFACE".U1_STA3_CAM_Calibrations."Calibrate laser".Outputs.Result <> 1)) OR ("DB16000_OPC_UA_TRIGGER_ALARM".CLIENT.U1_STA3_COAXIAL.ALARMS.CAM_START_LASER_CALIB_METHOD_WORKING_BLOCKED_A AND NOT "DB2120_MPP_ITC_IPC".RESET_FAULTS)) AND "DB7254_UNIT_01_STA_3_COAXIAL_ENABLE_DISABLE".ENABLED;
   "DB426_ALARMS_WARNINGS".UNIT_01.STATION_3_COAXIAL."716721" := "DB16000_OPC_UA_TRIGGER_ALARM".CLIENT.U1_STA3_COAXIAL.ALARMS.CAM_START_LASER_CALIB_METHOD_WORKING_BLOCKED_A;
END_REGION

REGION Network 28: UNIT 01 STATION 3 COAXIAL CAMERA START NOZZLE CALIBRATION METHOD CONNECTION ALARM
   // CAMBIAR BIT DE ERROR DEL METODO CORRECTO
   RUNG wire#powerrail
      Contact( "DB16212_METHODCALL_U01_STA3_CAM_NOZZLE_CALIBRATE_TRIGGER".Error )
      wire#w1
      Contact( "DB7254_UNIT_01_STA_3_COAXIAL_ENABLE_DISABLE".ENABLED )
      wire#w2
      Coil( "DB16000_OPC_UA_TRIGGER_ALARM".CLIENT.U1_STA3_COAXIAL.ALARMS.CAM_START_NOZZLE_CALIB_CONNECTION_A )
   END_RUNG
   RUNG wire#powerrail
      Contact( "DB16000_OPC_UA_TRIGGER_ALARM".CLIENT.U1_STA3_COAXIAL.ALARMS.CAM_START_NOZZLE_CALIB_CONNECTION_A )
      I_Contact( "DB2120_MPP_ITC_IPC".RESET_FAULTS )
   END_RUNG wire#w1
   RUNG wire#w2
      Coil( "DB426_ALARMS_WARNINGS".UNIT_01.STATION_3_COAXIAL."716728" )
   END_RUNG
   // the same network as SCL:
   "DB16000_OPC_UA_TRIGGER_ALARM".CLIENT.U1_STA3_COAXIAL.ALARMS.CAM_START_NOZZLE_CALIB_CONNECTION_A := ("DB16212_METHODCALL_U01_STA3_CAM_NOZZLE_CALIBRATE_TRIGGER".Error OR ("DB16000_OPC_UA_TRIGGER_ALARM".CLIENT.U1_STA3_COAXIAL.ALARMS.CAM_START_NOZZLE_CALIB_CONNECTION_A AND NOT "DB2120_MPP_ITC_IPC".RESET_FAULTS)) AND "DB7254_UNIT_01_STA_3_COAXIAL_ENABLE_DISABLE".ENABLED;
   "DB426_ALARMS_WARNINGS".UNIT_01.STATION_3_COAXIAL."716728" := "DB16000_OPC_UA_TRIGGER_ALARM".CLIENT.U1_STA3_COAXIAL.ALARMS.CAM_START_NOZZLE_CALIB_CONNECTION_A;
END_REGION

REGION Network 29: UNIT 01 STATION 3 COAXIAL CAMERA START NOZZLE CALIBRATION METHOD WORKING OR BLOCKED ALARM
   // CAMBIAR BIT DE DONE DEL METODO CORRECTO
   RUNG wire#powerrail
      Contact( "DB16212_METHODCALL_U01_STA3_CAM_NOZZLE_CALIBRATE_TRIGGER".Done )
      { S7_Templates := "SrcType := Int" } NE_Contact(in1 := "DB16002_U01_STA3_COAXIAL_CLIENT_INTERFACE".U1_STA3_CAM_Calibrations."Calibrate nozzle".Outputs.Result, in2 := 1)
      wire#w1
      Contact( "DB7254_UNIT_01_STA_3_COAXIAL_ENABLE_DISABLE".ENABLED )
      wire#w2
      Coil( "DB16000_OPC_UA_TRIGGER_ALARM".CLIENT.U1_STA3_COAXIAL.ALARMS.CAM_START_NOZZLE_CALIB_METHOD_WORKING_BLOCKED_A )
   END_RUNG
   RUNG wire#powerrail
      Contact( "DB16000_OPC_UA_TRIGGER_ALARM".CLIENT.U1_STA3_COAXIAL.ALARMS.CAM_START_NOZZLE_CALIB_METHOD_WORKING_BLOCKED_A )
      I_Contact( "DB2120_MPP_ITC_IPC".RESET_FAULTS )
   END_RUNG wire#w1
   RUNG wire#w2
      Coil( "DB426_ALARMS_WARNINGS".UNIT_01.STATION_3_COAXIAL."716729" )
   END_RUNG
   // the same network as SCL:
   "DB16000_OPC_UA_TRIGGER_ALARM".CLIENT.U1_STA3_COAXIAL.ALARMS.CAM_START_NOZZLE_CALIB_METHOD_WORKING_BLOCKED_A := (("DB16212_METHODCALL_U01_STA3_CAM_NOZZLE_CALIBRATE_TRIGGER".Done AND ("DB16002_U01_STA3_COAXIAL_CLIENT_INTERFACE".U1_STA3_CAM_Calibrations."Calibrate nozzle".Outputs.Result <> 1)) OR ("DB16000_OPC_UA_TRIGGER_ALARM".CLIENT.U1_STA3_COAXIAL.ALARMS.CAM_START_NOZZLE_CALIB_METHOD_WORKING_BLOCKED_A AND NOT "DB2120_MPP_ITC_IPC".RESET_FAULTS)) AND "DB7254_UNIT_01_STA_3_COAXIAL_ENABLE_DISABLE".ENABLED;
   "DB426_ALARMS_WARNINGS".UNIT_01.STATION_3_COAXIAL."716729" := "DB16000_OPC_UA_TRIGGER_ALARM".CLIENT.U1_STA3_COAXIAL.ALARMS.CAM_START_NOZZLE_CALIB_METHOD_WORKING_BLOCKED_A;
END_REGION

REGION Network 30: UNIT 01 STATION 3 COAXIAL CAMERA START JET CALIBRATION METHOD CONNECTION ALARM
   // CAMBIAR BIT DE ERROR DEL METODO CORRECTO
   RUNG wire#powerrail
      Contact( "DB16213_METHODCALL_U01_STA3_CAM_JET_CALIBRATE_TRIGGER".Error )
      wire#w1
      Contact( "DB7254_UNIT_01_STA_3_COAXIAL_ENABLE_DISABLE".ENABLED )
      wire#w2
      Coil( "DB16000_OPC_UA_TRIGGER_ALARM".CLIENT.U1_STA3_COAXIAL.ALARMS.CAM_START_JET_CALIB_CONNECTION_A )
   END_RUNG
   RUNG wire#powerrail
      Contact( "DB16000_OPC_UA_TRIGGER_ALARM".CLIENT.U1_STA3_COAXIAL.ALARMS.CAM_START_JET_CALIB_CONNECTION_A )
      I_Contact( "DB2120_MPP_ITC_IPC".RESET_FAULTS )
   END_RUNG wire#w1
   RUNG wire#w2
      Coil( "DB426_ALARMS_WARNINGS".UNIT_01.STATION_3_COAXIAL."716736" )
   END_RUNG
   // the same network as SCL:
   "DB16000_OPC_UA_TRIGGER_ALARM".CLIENT.U1_STA3_COAXIAL.ALARMS.CAM_START_JET_CALIB_CONNECTION_A := ("DB16213_METHODCALL_U01_STA3_CAM_JET_CALIBRATE_TRIGGER".Error OR ("DB16000_OPC_UA_TRIGGER_ALARM".CLIENT.U1_STA3_COAXIAL.ALARMS.CAM_START_JET_CALIB_CONNECTION_A AND NOT "DB2120_MPP_ITC_IPC".RESET_FAULTS)) AND "DB7254_UNIT_01_STA_3_COAXIAL_ENABLE_DISABLE".ENABLED;
   "DB426_ALARMS_WARNINGS".UNIT_01.STATION_3_COAXIAL."716736" := "DB16000_OPC_UA_TRIGGER_ALARM".CLIENT.U1_STA3_COAXIAL.ALARMS.CAM_START_JET_CALIB_CONNECTION_A;
END_REGION

REGION Network 31: UNIT 01 STATION 3 COAXIAL CAMERA START JET CALIBRATION METHOD WORKING OR BLOCKED ALARM
   // CAMBIAR BIT DE DONE DEL METODO CORRECTO
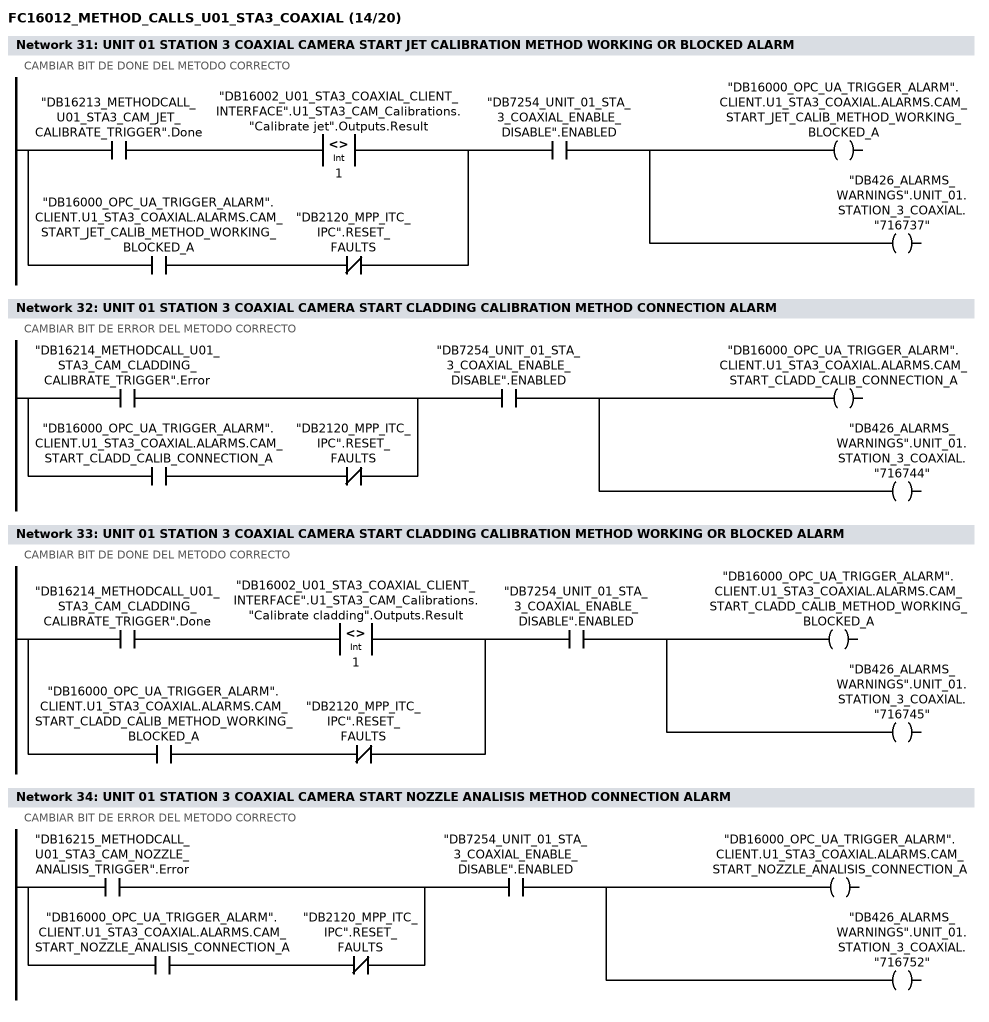
   RUNG wire#powerrail
      Contact( "DB16213_METHODCALL_U01_STA3_CAM_JET_CALIBRATE_TRIGGER".Done )
      { S7_Templates := "SrcType := Int" } NE_Contact(in1 := "DB16002_U01_STA3_COAXIAL_CLIENT_INTERFACE".U1_STA3_CAM_Calibrations."Calibrate jet".Outputs.Result, in2 := 1)
      wire#w1
      Contact( "DB7254_UNIT_01_STA_3_COAXIAL_ENABLE_DISABLE".ENABLED )
      wire#w2
      Coil( "DB16000_OPC_UA_TRIGGER_ALARM".CLIENT.U1_STA3_COAXIAL.ALARMS.CAM_START_JET_CALIB_METHOD_WORKING_BLOCKED_A )
   END_RUNG
   RUNG wire#powerrail
      Contact( "DB16000_OPC_UA_TRIGGER_ALARM".CLIENT.U1_STA3_COAXIAL.ALARMS.CAM_START_JET_CALIB_METHOD_WORKING_BLOCKED_A )
      I_Contact( "DB2120_MPP_ITC_IPC".RESET_FAULTS )
   END_RUNG wire#w1
   RUNG wire#w2
      Coil( "DB426_ALARMS_WARNINGS".UNIT_01.STATION_3_COAXIAL."716737" )
   END_RUNG
   // the same network as SCL:
   "DB16000_OPC_UA_TRIGGER_ALARM".CLIENT.U1_STA3_COAXIAL.ALARMS.CAM_START_JET_CALIB_METHOD_WORKING_BLOCKED_A := (("DB16213_METHODCALL_U01_STA3_CAM_JET_CALIBRATE_TRIGGER".Done AND ("DB16002_U01_STA3_COAXIAL_CLIENT_INTERFACE".U1_STA3_CAM_Calibrations."Calibrate jet".Outputs.Result <> 1)) OR ("DB16000_OPC_UA_TRIGGER_ALARM".CLIENT.U1_STA3_COAXIAL.ALARMS.CAM_START_JET_CALIB_METHOD_WORKING_BLOCKED_A AND NOT "DB2120_MPP_ITC_IPC".RESET_FAULTS)) AND "DB7254_UNIT_01_STA_3_COAXIAL_ENABLE_DISABLE".ENABLED;
   "DB426_ALARMS_WARNINGS".UNIT_01.STATION_3_COAXIAL."716737" := "DB16000_OPC_UA_TRIGGER_ALARM".CLIENT.U1_STA3_COAXIAL.ALARMS.CAM_START_JET_CALIB_METHOD_WORKING_BLOCKED_A;
END_REGION

REGION Network 32: UNIT 01 STATION 3 COAXIAL CAMERA START CLADDING CALIBRATION METHOD CONNECTION ALARM
   // CAMBIAR BIT DE ERROR DEL METODO CORRECTO
   RUNG wire#powerrail
      Contact( "DB16214_METHODCALL_U01_STA3_CAM_CLADDING_CALIBRATE_TRIGGER".Error )
      wire#w1
      Contact( "DB7254_UNIT_01_STA_3_COAXIAL_ENABLE_DISABLE".ENABLED )
      wire#w2
      Coil( "DB16000_OPC_UA_TRIGGER_ALARM".CLIENT.U1_STA3_COAXIAL.ALARMS.CAM_START_CLADD_CALIB_CONNECTION_A )
   END_RUNG
   RUNG wire#powerrail
      Contact( "DB16000_OPC_UA_TRIGGER_ALARM".CLIENT.U1_STA3_COAXIAL.ALARMS.CAM_START_CLADD_CALIB_CONNECTION_A )
      I_Contact( "DB2120_MPP_ITC_IPC".RESET_FAULTS )
   END_RUNG wire#w1
   RUNG wire#w2
      Coil( "DB426_ALARMS_WARNINGS".UNIT_01.STATION_3_COAXIAL."716744" )
   END_RUNG
   // the same network as SCL:
   "DB16000_OPC_UA_TRIGGER_ALARM".CLIENT.U1_STA3_COAXIAL.ALARMS.CAM_START_CLADD_CALIB_CONNECTION_A := ("DB16214_METHODCALL_U01_STA3_CAM_CLADDING_CALIBRATE_TRIGGER".Error OR ("DB16000_OPC_UA_TRIGGER_ALARM".CLIENT.U1_STA3_COAXIAL.ALARMS.CAM_START_CLADD_CALIB_CONNECTION_A AND NOT "DB2120_MPP_ITC_IPC".RESET_FAULTS)) AND "DB7254_UNIT_01_STA_3_COAXIAL_ENABLE_DISABLE".ENABLED;
   "DB426_ALARMS_WARNINGS".UNIT_01.STATION_3_COAXIAL."716744" := "DB16000_OPC_UA_TRIGGER_ALARM".CLIENT.U1_STA3_COAXIAL.ALARMS.CAM_START_CLADD_CALIB_CONNECTION_A;
END_REGION

REGION Network 33: UNIT 01 STATION 3 COAXIAL CAMERA START CLADDING CALIBRATION METHOD WORKING OR BLOCKED ALARM
   // CAMBIAR BIT DE DONE DEL METODO CORRECTO
   RUNG wire#powerrail
      Contact( "DB16214_METHODCALL_U01_STA3_CAM_CLADDING_CALIBRATE_TRIGGER".Done )
      { S7_Templates := "SrcType := Int" } NE_Contact(in1 := "DB16002_U01_STA3_COAXIAL_CLIENT_INTERFACE".U1_STA3_CAM_Calibrations."Calibrate cladding".Outputs.Result, in2 := 1)
      wire#w1
      Contact( "DB7254_UNIT_01_STA_3_COAXIAL_ENABLE_DISABLE".ENABLED )
      wire#w2
      Coil( "DB16000_OPC_UA_TRIGGER_ALARM".CLIENT.U1_STA3_COAXIAL.ALARMS.CAM_START_CLADD_CALIB_METHOD_WORKING_BLOCKED_A )
   END_RUNG
   RUNG wire#powerrail
      Contact( "DB16000_OPC_UA_TRIGGER_ALARM".CLIENT.U1_STA3_COAXIAL.ALARMS.CAM_START_CLADD_CALIB_METHOD_WORKING_BLOCKED_A )
      I_Contact( "DB2120_MPP_ITC_IPC".RESET_FAULTS )
   END_RUNG wire#w1
   RUNG wire#w2
      Coil( "DB426_ALARMS_WARNINGS".UNIT_01.STATION_3_COAXIAL."716745" )
   END_RUNG
   // the same network as SCL:
   "DB16000_OPC_UA_TRIGGER_ALARM".CLIENT.U1_STA3_COAXIAL.ALARMS.CAM_START_CLADD_CALIB_METHOD_WORKING_BLOCKED_A := (("DB16214_METHODCALL_U01_STA3_CAM_CLADDING_CALIBRATE_TRIGGER".Done AND ("DB16002_U01_STA3_COAXIAL_CLIENT_INTERFACE".U1_STA3_CAM_Calibrations."Calibrate cladding".Outputs.Result <> 1)) OR ("DB16000_OPC_UA_TRIGGER_ALARM".CLIENT.U1_STA3_COAXIAL.ALARMS.CAM_START_CLADD_CALIB_METHOD_WORKING_BLOCKED_A AND NOT "DB2120_MPP_ITC_IPC".RESET_FAULTS)) AND "DB7254_UNIT_01_STA_3_COAXIAL_ENABLE_DISABLE".ENABLED;
   "DB426_ALARMS_WARNINGS".UNIT_01.STATION_3_COAXIAL."716745" := "DB16000_OPC_UA_TRIGGER_ALARM".CLIENT.U1_STA3_COAXIAL.ALARMS.CAM_START_CLADD_CALIB_METHOD_WORKING_BLOCKED_A;
END_REGION

REGION Network 34: UNIT 01 STATION 3 COAXIAL CAMERA START NOZZLE ANALISIS METHOD CONNECTION ALARM
   // CAMBIAR BIT DE ERROR DEL METODO CORRECTO
   RUNG wire#powerrail
      Contact( "DB16215_METHODCALL_U01_STA3_CAM_NOZZLE_ANALISIS_TRIGGER".Error )
      wire#w1
      Contact( "DB7254_UNIT_01_STA_3_COAXIAL_ENABLE_DISABLE".ENABLED )
      wire#w2
      Coil( "DB16000_OPC_UA_TRIGGER_ALARM".CLIENT.U1_STA3_COAXIAL.ALARMS.CAM_START_NOZZLE_ANALISIS_CONNECTION_A )
   END_RUNG
   RUNG wire#powerrail
      Contact( "DB16000_OPC_UA_TRIGGER_ALARM".CLIENT.U1_STA3_COAXIAL.ALARMS.CAM_START_NOZZLE_ANALISIS_CONNECTION_A )
      I_Contact( "DB2120_MPP_ITC_IPC".RESET_FAULTS )
   END_RUNG wire#w1
   RUNG wire#w2
      Coil( "DB426_ALARMS_WARNINGS".UNIT_01.STATION_3_COAXIAL."716752" )
   END_RUNG
   // the same network as SCL:
   "DB16000_OPC_UA_TRIGGER_ALARM".CLIENT.U1_STA3_COAXIAL.ALARMS.CAM_START_NOZZLE_ANALISIS_CONNECTION_A := ("DB16215_METHODCALL_U01_STA3_CAM_NOZZLE_ANALISIS_TRIGGER".Error OR ("DB16000_OPC_UA_TRIGGER_ALARM".CLIENT.U1_STA3_COAXIAL.ALARMS.CAM_START_NOZZLE_ANALISIS_CONNECTION_A AND NOT "DB2120_MPP_ITC_IPC".RESET_FAULTS)) AND "DB7254_UNIT_01_STA_3_COAXIAL_ENABLE_DISABLE".ENABLED;
   "DB426_ALARMS_WARNINGS".UNIT_01.STATION_3_COAXIAL."716752" := "DB16000_OPC_UA_TRIGGER_ALARM".CLIENT.U1_STA3_COAXIAL.ALARMS.CAM_START_NOZZLE_ANALISIS_CONNECTION_A;
END_REGION

REGION Network 35: UNIT 01 STATION 3 COAXIAL CAMERA START NOZZLE ANALISIS METHOD WORKING OR BLOCKED ALARM
   // CAMBIAR BIT DE DONE DEL METODO CORRECTO
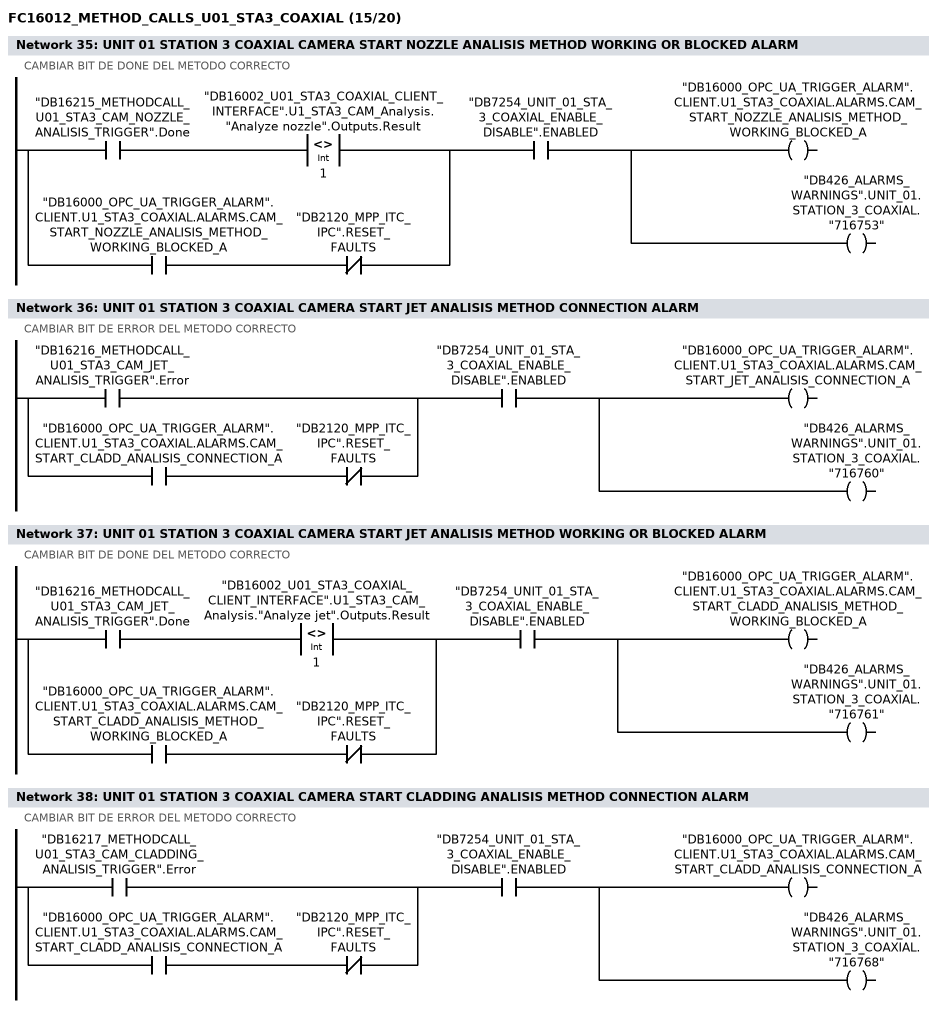
   RUNG wire#powerrail
      Contact( "DB16215_METHODCALL_U01_STA3_CAM_NOZZLE_ANALISIS_TRIGGER".Done )
      { S7_Templates := "SrcType := Int" } NE_Contact(in1 := "DB16002_U01_STA3_COAXIAL_CLIENT_INTERFACE".U1_STA3_CAM_Analysis."Analyze nozzle".Outputs.Result, in2 := 1)
      wire#w1
      Contact( "DB7254_UNIT_01_STA_3_COAXIAL_ENABLE_DISABLE".ENABLED )
      wire#w2
      Coil( "DB16000_OPC_UA_TRIGGER_ALARM".CLIENT.U1_STA3_COAXIAL.ALARMS.CAM_START_NOZZLE_ANALISIS_METHOD_WORKING_BLOCKED_A )
   END_RUNG
   RUNG wire#powerrail
      Contact( "DB16000_OPC_UA_TRIGGER_ALARM".CLIENT.U1_STA3_COAXIAL.ALARMS.CAM_START_NOZZLE_ANALISIS_METHOD_WORKING_BLOCKED_A )
      I_Contact( "DB2120_MPP_ITC_IPC".RESET_FAULTS )
   END_RUNG wire#w1
   RUNG wire#w2
      Coil( "DB426_ALARMS_WARNINGS".UNIT_01.STATION_3_COAXIAL."716753" )
   END_RUNG
   // the same network as SCL:
   "DB16000_OPC_UA_TRIGGER_ALARM".CLIENT.U1_STA3_COAXIAL.ALARMS.CAM_START_NOZZLE_ANALISIS_METHOD_WORKING_BLOCKED_A := (("DB16215_METHODCALL_U01_STA3_CAM_NOZZLE_ANALISIS_TRIGGER".Done AND ("DB16002_U01_STA3_COAXIAL_CLIENT_INTERFACE".U1_STA3_CAM_Analysis."Analyze nozzle".Outputs.Result <> 1)) OR ("DB16000_OPC_UA_TRIGGER_ALARM".CLIENT.U1_STA3_COAXIAL.ALARMS.CAM_START_NOZZLE_ANALISIS_METHOD_WORKING_BLOCKED_A AND NOT "DB2120_MPP_ITC_IPC".RESET_FAULTS)) AND "DB7254_UNIT_01_STA_3_COAXIAL_ENABLE_DISABLE".ENABLED;
   "DB426_ALARMS_WARNINGS".UNIT_01.STATION_3_COAXIAL."716753" := "DB16000_OPC_UA_TRIGGER_ALARM".CLIENT.U1_STA3_COAXIAL.ALARMS.CAM_START_NOZZLE_ANALISIS_METHOD_WORKING_BLOCKED_A;
END_REGION

REGION Network 36: UNIT 01 STATION 3 COAXIAL CAMERA START JET ANALISIS METHOD CONNECTION ALARM
   // CAMBIAR BIT DE ERROR DEL METODO CORRECTO
   RUNG wire#powerrail
      Contact( "DB16216_METHODCALL_U01_STA3_CAM_JET_ANALISIS_TRIGGER".Error )
      wire#w1
      Contact( "DB7254_UNIT_01_STA_3_COAXIAL_ENABLE_DISABLE".ENABLED )
      wire#w2
      Coil( "DB16000_OPC_UA_TRIGGER_ALARM".CLIENT.U1_STA3_COAXIAL.ALARMS.CAM_START_JET_ANALISIS_CONNECTION_A )
   END_RUNG
   RUNG wire#powerrail
      Contact( "DB16000_OPC_UA_TRIGGER_ALARM".CLIENT.U1_STA3_COAXIAL.ALARMS.CAM_START_CLADD_ANALISIS_CONNECTION_A )
      I_Contact( "DB2120_MPP_ITC_IPC".RESET_FAULTS )
   END_RUNG wire#w1
   RUNG wire#w2
      Coil( "DB426_ALARMS_WARNINGS".UNIT_01.STATION_3_COAXIAL."716760" )
   END_RUNG
   // the same network as SCL:
   "DB16000_OPC_UA_TRIGGER_ALARM".CLIENT.U1_STA3_COAXIAL.ALARMS.CAM_START_JET_ANALISIS_CONNECTION_A := ("DB16216_METHODCALL_U01_STA3_CAM_JET_ANALISIS_TRIGGER".Error OR ("DB16000_OPC_UA_TRIGGER_ALARM".CLIENT.U1_STA3_COAXIAL.ALARMS.CAM_START_CLADD_ANALISIS_CONNECTION_A AND NOT "DB2120_MPP_ITC_IPC".RESET_FAULTS)) AND "DB7254_UNIT_01_STA_3_COAXIAL_ENABLE_DISABLE".ENABLED;
   "DB426_ALARMS_WARNINGS".UNIT_01.STATION_3_COAXIAL."716760" := "DB16000_OPC_UA_TRIGGER_ALARM".CLIENT.U1_STA3_COAXIAL.ALARMS.CAM_START_JET_ANALISIS_CONNECTION_A;
END_REGION

REGION Network 37: UNIT 01 STATION 3 COAXIAL CAMERA START JET ANALISIS METHOD WORKING OR BLOCKED ALARM
   // CAMBIAR BIT DE DONE DEL METODO CORRECTO
   RUNG wire#powerrail
      Contact( "DB16216_METHODCALL_U01_STA3_CAM_JET_ANALISIS_TRIGGER".Done )
      { S7_Templates := "SrcType := Int" } NE_Contact(in1 := "DB16002_U01_STA3_COAXIAL_CLIENT_INTERFACE".U1_STA3_CAM_Analysis."Analyze jet".Outputs.Result, in2 := 1)
      wire#w1
      Contact( "DB7254_UNIT_01_STA_3_COAXIAL_ENABLE_DISABLE".ENABLED )
      wire#w2
      Coil( "DB16000_OPC_UA_TRIGGER_ALARM".CLIENT.U1_STA3_COAXIAL.ALARMS.CAM_START_CLADD_ANALISIS_METHOD_WORKING_BLOCKED_A )
   END_RUNG
   RUNG wire#powerrail
      Contact( "DB16000_OPC_UA_TRIGGER_ALARM".CLIENT.U1_STA3_COAXIAL.ALARMS.CAM_START_CLADD_ANALISIS_METHOD_WORKING_BLOCKED_A )
      I_Contact( "DB2120_MPP_ITC_IPC".RESET_FAULTS )
   END_RUNG wire#w1
   RUNG wire#w2
      Coil( "DB426_ALARMS_WARNINGS".UNIT_01.STATION_3_COAXIAL."716761" )
   END_RUNG
   // the same network as SCL:
   "DB16000_OPC_UA_TRIGGER_ALARM".CLIENT.U1_STA3_COAXIAL.ALARMS.CAM_START_CLADD_ANALISIS_METHOD_WORKING_BLOCKED_A := (("DB16216_METHODCALL_U01_STA3_CAM_JET_ANALISIS_TRIGGER".Done AND ("DB16002_U01_STA3_COAXIAL_CLIENT_INTERFACE".U1_STA3_CAM_Analysis."Analyze jet".Outputs.Result <> 1)) OR ("DB16000_OPC_UA_TRIGGER_ALARM".CLIENT.U1_STA3_COAXIAL.ALARMS.CAM_START_CLADD_ANALISIS_METHOD_WORKING_BLOCKED_A AND NOT "DB2120_MPP_ITC_IPC".RESET_FAULTS)) AND "DB7254_UNIT_01_STA_3_COAXIAL_ENABLE_DISABLE".ENABLED;
   "DB426_ALARMS_WARNINGS".UNIT_01.STATION_3_COAXIAL."716761" := "DB16000_OPC_UA_TRIGGER_ALARM".CLIENT.U1_STA3_COAXIAL.ALARMS.CAM_START_CLADD_ANALISIS_METHOD_WORKING_BLOCKED_A;
END_REGION

REGION Network 38: UNIT 01 STATION 3 COAXIAL CAMERA START CLADDING ANALISIS METHOD CONNECTION ALARM
   // CAMBIAR BIT DE ERROR DEL METODO CORRECTO
   RUNG wire#powerrail
      Contact( "DB16217_METHODCALL_U01_STA3_CAM_CLADDING_ANALISIS_TRIGGER".Error )
      wire#w1
      Contact( "DB7254_UNIT_01_STA_3_COAXIAL_ENABLE_DISABLE".ENABLED )
      wire#w2
      Coil( "DB16000_OPC_UA_TRIGGER_ALARM".CLIENT.U1_STA3_COAXIAL.ALARMS.CAM_START_CLADD_ANALISIS_CONNECTION_A )
   END_RUNG
   RUNG wire#powerrail
      Contact( "DB16000_OPC_UA_TRIGGER_ALARM".CLIENT.U1_STA3_COAXIAL.ALARMS.CAM_START_CLADD_ANALISIS_CONNECTION_A )
      I_Contact( "DB2120_MPP_ITC_IPC".RESET_FAULTS )
   END_RUNG wire#w1
   RUNG wire#w2
      Coil( "DB426_ALARMS_WARNINGS".UNIT_01.STATION_3_COAXIAL."716768" )
   END_RUNG
   // the same network as SCL:
   "DB16000_OPC_UA_TRIGGER_ALARM".CLIENT.U1_STA3_COAXIAL.ALARMS.CAM_START_CLADD_ANALISIS_CONNECTION_A := ("DB16217_METHODCALL_U01_STA3_CAM_CLADDING_ANALISIS_TRIGGER".Error OR ("DB16000_OPC_UA_TRIGGER_ALARM".CLIENT.U1_STA3_COAXIAL.ALARMS.CAM_START_CLADD_ANALISIS_CONNECTION_A AND NOT "DB2120_MPP_ITC_IPC".RESET_FAULTS)) AND "DB7254_UNIT_01_STA_3_COAXIAL_ENABLE_DISABLE".ENABLED;
   "DB426_ALARMS_WARNINGS".UNIT_01.STATION_3_COAXIAL."716768" := "DB16000_OPC_UA_TRIGGER_ALARM".CLIENT.U1_STA3_COAXIAL.ALARMS.CAM_START_CLADD_ANALISIS_CONNECTION_A;
END_REGION

REGION Network 39: UNIT 01 STATION 3 COAXIAL CAMERA START CLADDING ANALISIS METHOD WORKING OR BLOCKED ALARM
   // CAMBIAR BIT DE DONE DEL METODO CORRECTO
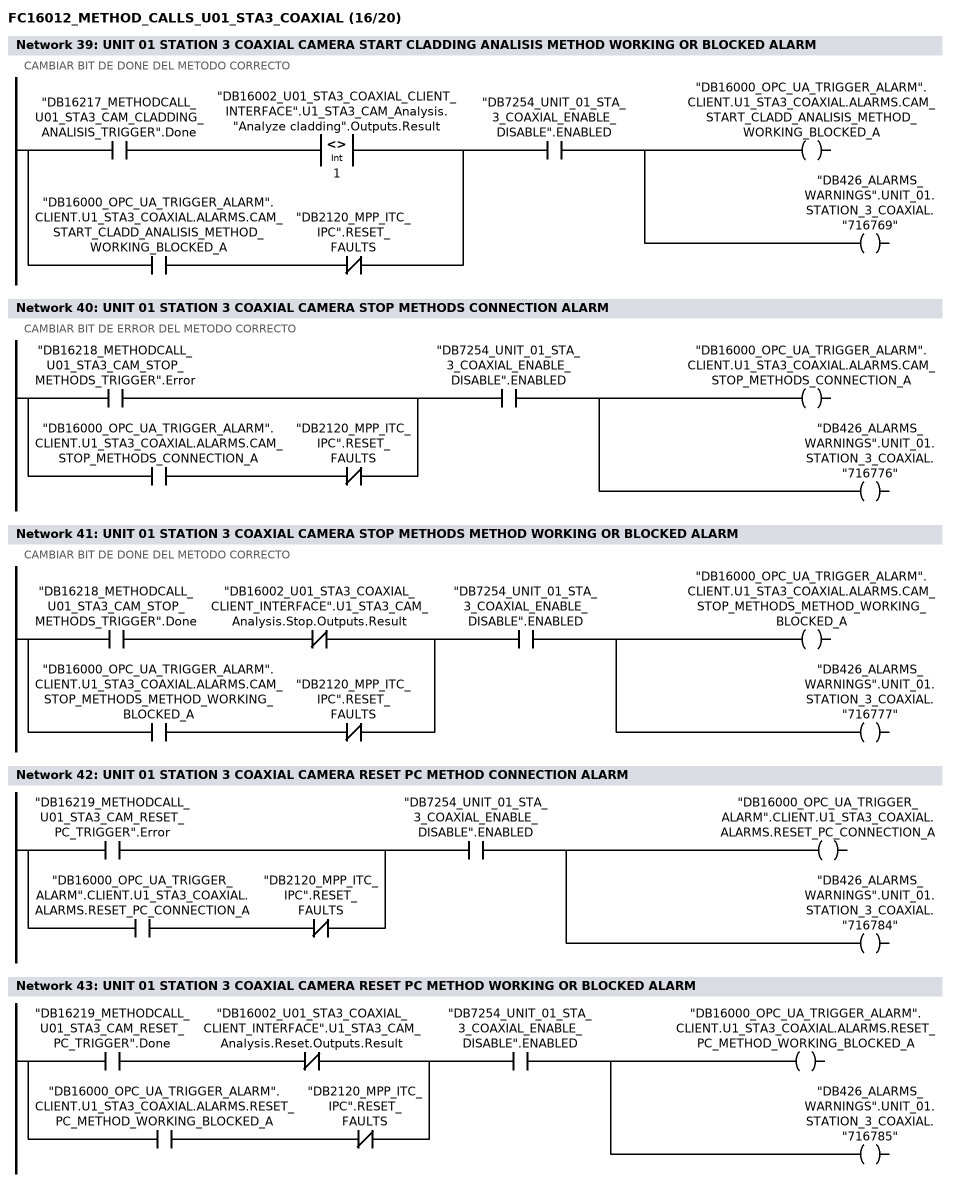
   RUNG wire#powerrail
      Contact( "DB16217_METHODCALL_U01_STA3_CAM_CLADDING_ANALISIS_TRIGGER".Done )
      { S7_Templates := "SrcType := Int" } NE_Contact(in1 := "DB16002_U01_STA3_COAXIAL_CLIENT_INTERFACE".U1_STA3_CAM_Analysis."Analyze cladding".Outputs.Result, in2 := 1)
      wire#w1
      Contact( "DB7254_UNIT_01_STA_3_COAXIAL_ENABLE_DISABLE".ENABLED )
      wire#w2
      Coil( "DB16000_OPC_UA_TRIGGER_ALARM".CLIENT.U1_STA3_COAXIAL.ALARMS.CAM_START_CLADD_ANALISIS_METHOD_WORKING_BLOCKED_A )
   END_RUNG
   RUNG wire#powerrail
      Contact( "DB16000_OPC_UA_TRIGGER_ALARM".CLIENT.U1_STA3_COAXIAL.ALARMS.CAM_START_CLADD_ANALISIS_METHOD_WORKING_BLOCKED_A )
      I_Contact( "DB2120_MPP_ITC_IPC".RESET_FAULTS )
   END_RUNG wire#w1
   RUNG wire#w2
      Coil( "DB426_ALARMS_WARNINGS".UNIT_01.STATION_3_COAXIAL."716769" )
   END_RUNG
   // the same network as SCL:
   "DB16000_OPC_UA_TRIGGER_ALARM".CLIENT.U1_STA3_COAXIAL.ALARMS.CAM_START_CLADD_ANALISIS_METHOD_WORKING_BLOCKED_A := (("DB16217_METHODCALL_U01_STA3_CAM_CLADDING_ANALISIS_TRIGGER".Done AND ("DB16002_U01_STA3_COAXIAL_CLIENT_INTERFACE".U1_STA3_CAM_Analysis."Analyze cladding".Outputs.Result <> 1)) OR ("DB16000_OPC_UA_TRIGGER_ALARM".CLIENT.U1_STA3_COAXIAL.ALARMS.CAM_START_CLADD_ANALISIS_METHOD_WORKING_BLOCKED_A AND NOT "DB2120_MPP_ITC_IPC".RESET_FAULTS)) AND "DB7254_UNIT_01_STA_3_COAXIAL_ENABLE_DISABLE".ENABLED;
   "DB426_ALARMS_WARNINGS".UNIT_01.STATION_3_COAXIAL."716769" := "DB16000_OPC_UA_TRIGGER_ALARM".CLIENT.U1_STA3_COAXIAL.ALARMS.CAM_START_CLADD_ANALISIS_METHOD_WORKING_BLOCKED_A;
END_REGION

REGION Network 40: UNIT 01 STATION 3 COAXIAL CAMERA STOP METHODS CONNECTION ALARM
   // CAMBIAR BIT DE ERROR DEL METODO CORRECTO
   RUNG wire#powerrail
      Contact( "DB16218_METHODCALL_U01_STA3_CAM_STOP_METHODS_TRIGGER".Error )
      wire#w1
      Contact( "DB7254_UNIT_01_STA_3_COAXIAL_ENABLE_DISABLE".ENABLED )
      wire#w2
      Coil( "DB16000_OPC_UA_TRIGGER_ALARM".CLIENT.U1_STA3_COAXIAL.ALARMS.CAM_STOP_METHODS_CONNECTION_A )
   END_RUNG
   RUNG wire#powerrail
      Contact( "DB16000_OPC_UA_TRIGGER_ALARM".CLIENT.U1_STA3_COAXIAL.ALARMS.CAM_STOP_METHODS_CONNECTION_A )
      I_Contact( "DB2120_MPP_ITC_IPC".RESET_FAULTS )
   END_RUNG wire#w1
   RUNG wire#w2
      Coil( "DB426_ALARMS_WARNINGS".UNIT_01.STATION_3_COAXIAL."716776" )
   END_RUNG
   // the same network as SCL:
   "DB16000_OPC_UA_TRIGGER_ALARM".CLIENT.U1_STA3_COAXIAL.ALARMS.CAM_STOP_METHODS_CONNECTION_A := ("DB16218_METHODCALL_U01_STA3_CAM_STOP_METHODS_TRIGGER".Error OR ("DB16000_OPC_UA_TRIGGER_ALARM".CLIENT.U1_STA3_COAXIAL.ALARMS.CAM_STOP_METHODS_CONNECTION_A AND NOT "DB2120_MPP_ITC_IPC".RESET_FAULTS)) AND "DB7254_UNIT_01_STA_3_COAXIAL_ENABLE_DISABLE".ENABLED;
   "DB426_ALARMS_WARNINGS".UNIT_01.STATION_3_COAXIAL."716776" := "DB16000_OPC_UA_TRIGGER_ALARM".CLIENT.U1_STA3_COAXIAL.ALARMS.CAM_STOP_METHODS_CONNECTION_A;
END_REGION

REGION Network 41: UNIT 01 STATION 3 COAXIAL CAMERA STOP METHODS METHOD WORKING OR BLOCKED ALARM
   // CAMBIAR BIT DE DONE DEL METODO CORRECTO
   RUNG wire#powerrail
      Contact( "DB16218_METHODCALL_U01_STA3_CAM_STOP_METHODS_TRIGGER".Done )
      I_Contact( "DB16002_U01_STA3_COAXIAL_CLIENT_INTERFACE".U1_STA3_CAM_Analysis.Stop.Outputs.Result )
      wire#w1
      Contact( "DB7254_UNIT_01_STA_3_COAXIAL_ENABLE_DISABLE".ENABLED )
      wire#w2
      Coil( "DB16000_OPC_UA_TRIGGER_ALARM".CLIENT.U1_STA3_COAXIAL.ALARMS.CAM_STOP_METHODS_METHOD_WORKING_BLOCKED_A )
   END_RUNG
   RUNG wire#powerrail
      Contact( "DB16000_OPC_UA_TRIGGER_ALARM".CLIENT.U1_STA3_COAXIAL.ALARMS.CAM_STOP_METHODS_METHOD_WORKING_BLOCKED_A )
      I_Contact( "DB2120_MPP_ITC_IPC".RESET_FAULTS )
   END_RUNG wire#w1
   RUNG wire#w2
      Coil( "DB426_ALARMS_WARNINGS".UNIT_01.STATION_3_COAXIAL."716777" )
   END_RUNG
   // the same network as SCL:
   "DB16000_OPC_UA_TRIGGER_ALARM".CLIENT.U1_STA3_COAXIAL.ALARMS.CAM_STOP_METHODS_METHOD_WORKING_BLOCKED_A := (("DB16218_METHODCALL_U01_STA3_CAM_STOP_METHODS_TRIGGER".Done AND NOT "DB16002_U01_STA3_COAXIAL_CLIENT_INTERFACE".U1_STA3_CAM_Analysis.Stop.Outputs.Result) OR ("DB16000_OPC_UA_TRIGGER_ALARM".CLIENT.U1_STA3_COAXIAL.ALARMS.CAM_STOP_METHODS_METHOD_WORKING_BLOCKED_A AND NOT "DB2120_MPP_ITC_IPC".RESET_FAULTS)) AND "DB7254_UNIT_01_STA_3_COAXIAL_ENABLE_DISABLE".ENABLED;
   "DB426_ALARMS_WARNINGS".UNIT_01.STATION_3_COAXIAL."716777" := "DB16000_OPC_UA_TRIGGER_ALARM".CLIENT.U1_STA3_COAXIAL.ALARMS.CAM_STOP_METHODS_METHOD_WORKING_BLOCKED_A;
END_REGION

REGION Network 42: UNIT 01 STATION 3 COAXIAL CAMERA RESET PC METHOD CONNECTION ALARM
   RUNG wire#powerrail
      Contact( "DB16219_METHODCALL_U01_STA3_CAM_RESET_PC_TRIGGER".Error )
      wire#w1
      Contact( "DB7254_UNIT_01_STA_3_COAXIAL_ENABLE_DISABLE".ENABLED )
      wire#w2
      Coil( "DB16000_OPC_UA_TRIGGER_ALARM".CLIENT.U1_STA3_COAXIAL.ALARMS.RESET_PC_CONNECTION_A )
   END_RUNG
   RUNG wire#powerrail
      Contact( "DB16000_OPC_UA_TRIGGER_ALARM".CLIENT.U1_STA3_COAXIAL.ALARMS.RESET_PC_CONNECTION_A )
      I_Contact( "DB2120_MPP_ITC_IPC".RESET_FAULTS )
   END_RUNG wire#w1
   RUNG wire#w2
      Coil( "DB426_ALARMS_WARNINGS".UNIT_01.STATION_3_COAXIAL."716784" )
   END_RUNG
   // the same network as SCL:
   "DB16000_OPC_UA_TRIGGER_ALARM".CLIENT.U1_STA3_COAXIAL.ALARMS.RESET_PC_CONNECTION_A := ("DB16219_METHODCALL_U01_STA3_CAM_RESET_PC_TRIGGER".Error OR ("DB16000_OPC_UA_TRIGGER_ALARM".CLIENT.U1_STA3_COAXIAL.ALARMS.RESET_PC_CONNECTION_A AND NOT "DB2120_MPP_ITC_IPC".RESET_FAULTS)) AND "DB7254_UNIT_01_STA_3_COAXIAL_ENABLE_DISABLE".ENABLED;
   "DB426_ALARMS_WARNINGS".UNIT_01.STATION_3_COAXIAL."716784" := "DB16000_OPC_UA_TRIGGER_ALARM".CLIENT.U1_STA3_COAXIAL.ALARMS.RESET_PC_CONNECTION_A;
END_REGION

REGION Network 43: UNIT 01 STATION 3 COAXIAL CAMERA RESET PC METHOD WORKING OR BLOCKED ALARM
   RUNG wire#powerrail
      Contact( "DB16219_METHODCALL_U01_STA3_CAM_RESET_PC_TRIGGER".Done )
      I_Contact( "DB16002_U01_STA3_COAXIAL_CLIENT_INTERFACE".U1_STA3_CAM_Analysis.Reset.Outputs.Result )
      wire#w1
      Contact( "DB7254_UNIT_01_STA_3_COAXIAL_ENABLE_DISABLE".ENABLED )
      wire#w2
      Coil( "DB16000_OPC_UA_TRIGGER_ALARM".CLIENT.U1_STA3_COAXIAL.ALARMS.RESET_PC_METHOD_WORKING_BLOCKED_A )
   END_RUNG
   RUNG wire#powerrail
      Contact( "DB16000_OPC_UA_TRIGGER_ALARM".CLIENT.U1_STA3_COAXIAL.ALARMS.RESET_PC_METHOD_WORKING_BLOCKED_A )
      I_Contact( "DB2120_MPP_ITC_IPC".RESET_FAULTS )
   END_RUNG wire#w1
   RUNG wire#w2
      Coil( "DB426_ALARMS_WARNINGS".UNIT_01.STATION_3_COAXIAL."716785" )
   END_RUNG
   // the same network as SCL:
   "DB16000_OPC_UA_TRIGGER_ALARM".CLIENT.U1_STA3_COAXIAL.ALARMS.RESET_PC_METHOD_WORKING_BLOCKED_A := (("DB16219_METHODCALL_U01_STA3_CAM_RESET_PC_TRIGGER".Done AND NOT "DB16002_U01_STA3_COAXIAL_CLIENT_INTERFACE".U1_STA3_CAM_Analysis.Reset.Outputs.Result) OR ("DB16000_OPC_UA_TRIGGER_ALARM".CLIENT.U1_STA3_COAXIAL.ALARMS.RESET_PC_METHOD_WORKING_BLOCKED_A AND NOT "DB2120_MPP_ITC_IPC".RESET_FAULTS)) AND "DB7254_UNIT_01_STA_3_COAXIAL_ENABLE_DISABLE".ENABLED;
   "DB426_ALARMS_WARNINGS".UNIT_01.STATION_3_COAXIAL."716785" := "DB16000_OPC_UA_TRIGGER_ALARM".CLIENT.U1_STA3_COAXIAL.ALARMS.RESET_PC_METHOD_WORKING_BLOCKED_A;
END_REGION

REGION Network 44: UNIT 01 STATION 3 COAXIAL CAMERA READ VARIABLES METHOD CONNECTION ALARM
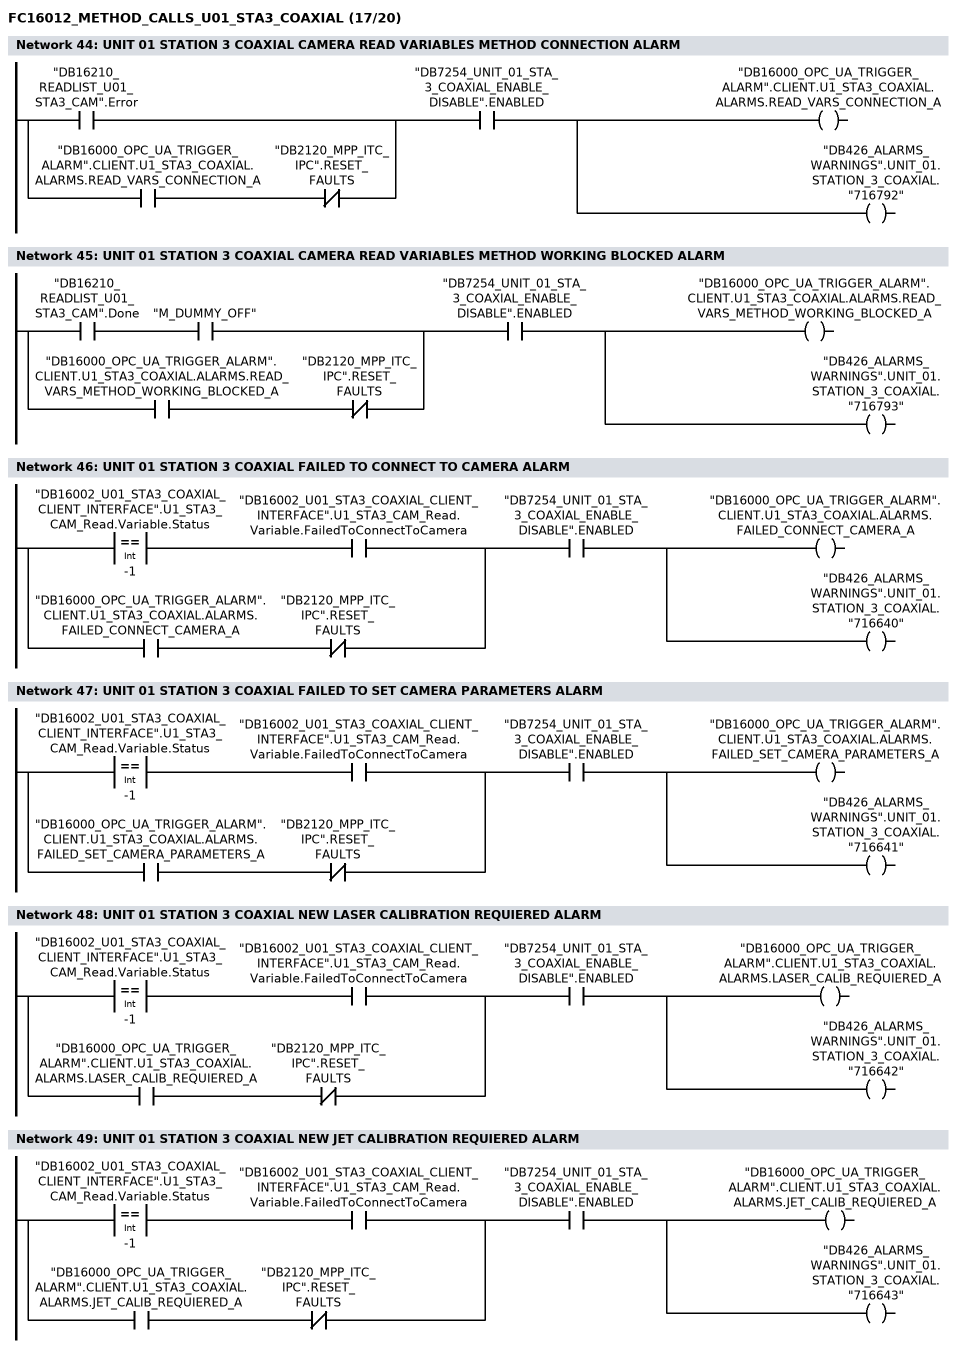
   RUNG wire#powerrail
      Contact( "DB16210_READLIST_U01_STA3_CAM".Error )
      wire#w1
      Contact( "DB7254_UNIT_01_STA_3_COAXIAL_ENABLE_DISABLE".ENABLED )
      wire#w2
      Coil( "DB16000_OPC_UA_TRIGGER_ALARM".CLIENT.U1_STA3_COAXIAL.ALARMS.READ_VARS_CONNECTION_A )
   END_RUNG
   RUNG wire#powerrail
      Contact( "DB16000_OPC_UA_TRIGGER_ALARM".CLIENT.U1_STA3_COAXIAL.ALARMS.READ_VARS_CONNECTION_A )
      I_Contact( "DB2120_MPP_ITC_IPC".RESET_FAULTS )
   END_RUNG wire#w1
   RUNG wire#w2
      Coil( "DB426_ALARMS_WARNINGS".UNIT_01.STATION_3_COAXIAL."716792" )
   END_RUNG
   // the same network as SCL:
   "DB16000_OPC_UA_TRIGGER_ALARM".CLIENT.U1_STA3_COAXIAL.ALARMS.READ_VARS_CONNECTION_A := ("DB16210_READLIST_U01_STA3_CAM".Error OR ("DB16000_OPC_UA_TRIGGER_ALARM".CLIENT.U1_STA3_COAXIAL.ALARMS.READ_VARS_CONNECTION_A AND NOT "DB2120_MPP_ITC_IPC".RESET_FAULTS)) AND "DB7254_UNIT_01_STA_3_COAXIAL_ENABLE_DISABLE".ENABLED;
   "DB426_ALARMS_WARNINGS".UNIT_01.STATION_3_COAXIAL."716792" := "DB16000_OPC_UA_TRIGGER_ALARM".CLIENT.U1_STA3_COAXIAL.ALARMS.READ_VARS_CONNECTION_A;
END_REGION

REGION Network 45: UNIT 01 STATION 3 COAXIAL CAMERA READ VARIABLES METHOD WORKING BLOCKED ALARM
   RUNG wire#powerrail
      Contact( "DB16210_READLIST_U01_STA3_CAM".Done )
      Contact( "M_DUMMY_OFF" )
      wire#w1
      Contact( "DB7254_UNIT_01_STA_3_COAXIAL_ENABLE_DISABLE".ENABLED )
      wire#w2
      Coil( "DB16000_OPC_UA_TRIGGER_ALARM".CLIENT.U1_STA3_COAXIAL.ALARMS.READ_VARS_METHOD_WORKING_BLOCKED_A )
   END_RUNG
   RUNG wire#powerrail
      Contact( "DB16000_OPC_UA_TRIGGER_ALARM".CLIENT.U1_STA3_COAXIAL.ALARMS.READ_VARS_METHOD_WORKING_BLOCKED_A )
      I_Contact( "DB2120_MPP_ITC_IPC".RESET_FAULTS )
   END_RUNG wire#w1
   RUNG wire#w2
      Coil( "DB426_ALARMS_WARNINGS".UNIT_01.STATION_3_COAXIAL."716793" )
   END_RUNG
   // the same network as SCL:
   "DB16000_OPC_UA_TRIGGER_ALARM".CLIENT.U1_STA3_COAXIAL.ALARMS.READ_VARS_METHOD_WORKING_BLOCKED_A := (("DB16210_READLIST_U01_STA3_CAM".Done AND "M_DUMMY_OFF") OR ("DB16000_OPC_UA_TRIGGER_ALARM".CLIENT.U1_STA3_COAXIAL.ALARMS.READ_VARS_METHOD_WORKING_BLOCKED_A AND NOT "DB2120_MPP_ITC_IPC".RESET_FAULTS)) AND "DB7254_UNIT_01_STA_3_COAXIAL_ENABLE_DISABLE".ENABLED;
   "DB426_ALARMS_WARNINGS".UNIT_01.STATION_3_COAXIAL."716793" := "DB16000_OPC_UA_TRIGGER_ALARM".CLIENT.U1_STA3_COAXIAL.ALARMS.READ_VARS_METHOD_WORKING_BLOCKED_A;
END_REGION

REGION Network 46: UNIT 01 STATION 3 COAXIAL FAILED TO CONNECT TO CAMERA ALARM
   RUNG wire#powerrail
      { S7_Templates := "SrcType := Int" } EQ_Contact(in1 := "DB16002_U01_STA3_COAXIAL_CLIENT_INTERFACE".U1_STA3_CAM_Read.Variable.Status, in2 := -1)
      Contact( "DB16002_U01_STA3_COAXIAL_CLIENT_INTERFACE".U1_STA3_CAM_Read.Variable.FailedToConnectToCamera )
      wire#w1
      Contact( "DB7254_UNIT_01_STA_3_COAXIAL_ENABLE_DISABLE".ENABLED )
      wire#w2
      Coil( "DB16000_OPC_UA_TRIGGER_ALARM".CLIENT.U1_STA3_COAXIAL.ALARMS.FAILED_CONNECT_CAMERA_A )
   END_RUNG
   RUNG wire#powerrail
      Contact( "DB16000_OPC_UA_TRIGGER_ALARM".CLIENT.U1_STA3_COAXIAL.ALARMS.FAILED_CONNECT_CAMERA_A )
      I_Contact( "DB2120_MPP_ITC_IPC".RESET_FAULTS )
   END_RUNG wire#w1
   RUNG wire#w2
      Coil( "DB426_ALARMS_WARNINGS".UNIT_01.STATION_3_COAXIAL."716640" )
   END_RUNG
   // the same network as SCL:
   "DB16000_OPC_UA_TRIGGER_ALARM".CLIENT.U1_STA3_COAXIAL.ALARMS.FAILED_CONNECT_CAMERA_A := ((("DB16002_U01_STA3_COAXIAL_CLIENT_INTERFACE".U1_STA3_CAM_Read.Variable.Status = (-1)) AND "DB16002_U01_STA3_COAXIAL_CLIENT_INTERFACE".U1_STA3_CAM_Read.Variable.FailedToConnectToCamera) OR ("DB16000_OPC_UA_TRIGGER_ALARM".CLIENT.U1_STA3_COAXIAL.ALARMS.FAILED_CONNECT_CAMERA_A AND NOT "DB2120_MPP_ITC_IPC".RESET_FAULTS)) AND "DB7254_UNIT_01_STA_3_COAXIAL_ENABLE_DISABLE".ENABLED;
   "DB426_ALARMS_WARNINGS".UNIT_01.STATION_3_COAXIAL."716640" := "DB16000_OPC_UA_TRIGGER_ALARM".CLIENT.U1_STA3_COAXIAL.ALARMS.FAILED_CONNECT_CAMERA_A;
END_REGION

REGION Network 47: UNIT 01 STATION 3 COAXIAL FAILED TO SET CAMERA PARAMETERS ALARM
   RUNG wire#powerrail
      { S7_Templates := "SrcType := Int" } EQ_Contact(in1 := "DB16002_U01_STA3_COAXIAL_CLIENT_INTERFACE".U1_STA3_CAM_Read.Variable.Status, in2 := -1)
      Contact( "DB16002_U01_STA3_COAXIAL_CLIENT_INTERFACE".U1_STA3_CAM_Read.Variable.FailedToConnectToCamera )
      wire#w1
      Contact( "DB7254_UNIT_01_STA_3_COAXIAL_ENABLE_DISABLE".ENABLED )
      wire#w2
      Coil( "DB16000_OPC_UA_TRIGGER_ALARM".CLIENT.U1_STA3_COAXIAL.ALARMS.FAILED_SET_CAMERA_PARAMETERS_A )
   END_RUNG
   RUNG wire#powerrail
      Contact( "DB16000_OPC_UA_TRIGGER_ALARM".CLIENT.U1_STA3_COAXIAL.ALARMS.FAILED_SET_CAMERA_PARAMETERS_A )
      I_Contact( "DB2120_MPP_ITC_IPC".RESET_FAULTS )
   END_RUNG wire#w1
   RUNG wire#w2
      Coil( "DB426_ALARMS_WARNINGS".UNIT_01.STATION_3_COAXIAL."716641" )
   END_RUNG
   // the same network as SCL:
   "DB16000_OPC_UA_TRIGGER_ALARM".CLIENT.U1_STA3_COAXIAL.ALARMS.FAILED_SET_CAMERA_PARAMETERS_A := ((("DB16002_U01_STA3_COAXIAL_CLIENT_INTERFACE".U1_STA3_CAM_Read.Variable.Status = (-1)) AND "DB16002_U01_STA3_COAXIAL_CLIENT_INTERFACE".U1_STA3_CAM_Read.Variable.FailedToConnectToCamera) OR ("DB16000_OPC_UA_TRIGGER_ALARM".CLIENT.U1_STA3_COAXIAL.ALARMS.FAILED_SET_CAMERA_PARAMETERS_A AND NOT "DB2120_MPP_ITC_IPC".RESET_FAULTS)) AND "DB7254_UNIT_01_STA_3_COAXIAL_ENABLE_DISABLE".ENABLED;
   "DB426_ALARMS_WARNINGS".UNIT_01.STATION_3_COAXIAL."716641" := "DB16000_OPC_UA_TRIGGER_ALARM".CLIENT.U1_STA3_COAXIAL.ALARMS.FAILED_SET_CAMERA_PARAMETERS_A;
END_REGION

REGION Network 48: UNIT 01 STATION 3 COAXIAL NEW LASER CALIBRATION REQUIERED ALARM
   RUNG wire#powerrail
      { S7_Templates := "SrcType := Int" } EQ_Contact(in1 := "DB16002_U01_STA3_COAXIAL_CLIENT_INTERFACE".U1_STA3_CAM_Read.Variable.Status, in2 := -1)
      Contact( "DB16002_U01_STA3_COAXIAL_CLIENT_INTERFACE".U1_STA3_CAM_Read.Variable.FailedToConnectToCamera )
      wire#w1
      Contact( "DB7254_UNIT_01_STA_3_COAXIAL_ENABLE_DISABLE".ENABLED )
      wire#w2
      Coil( "DB16000_OPC_UA_TRIGGER_ALARM".CLIENT.U1_STA3_COAXIAL.ALARMS.LASER_CALIB_REQUIERED_A )
   END_RUNG
   RUNG wire#powerrail
      Contact( "DB16000_OPC_UA_TRIGGER_ALARM".CLIENT.U1_STA3_COAXIAL.ALARMS.LASER_CALIB_REQUIERED_A )
      I_Contact( "DB2120_MPP_ITC_IPC".RESET_FAULTS )
   END_RUNG wire#w1
   RUNG wire#w2
      Coil( "DB426_ALARMS_WARNINGS".UNIT_01.STATION_3_COAXIAL."716642" )
   END_RUNG
   // the same network as SCL:
   "DB16000_OPC_UA_TRIGGER_ALARM".CLIENT.U1_STA3_COAXIAL.ALARMS.LASER_CALIB_REQUIERED_A := ((("DB16002_U01_STA3_COAXIAL_CLIENT_INTERFACE".U1_STA3_CAM_Read.Variable.Status = (-1)) AND "DB16002_U01_STA3_COAXIAL_CLIENT_INTERFACE".U1_STA3_CAM_Read.Variable.FailedToConnectToCamera) OR ("DB16000_OPC_UA_TRIGGER_ALARM".CLIENT.U1_STA3_COAXIAL.ALARMS.LASER_CALIB_REQUIERED_A AND NOT "DB2120_MPP_ITC_IPC".RESET_FAULTS)) AND "DB7254_UNIT_01_STA_3_COAXIAL_ENABLE_DISABLE".ENABLED;
   "DB426_ALARMS_WARNINGS".UNIT_01.STATION_3_COAXIAL."716642" := "DB16000_OPC_UA_TRIGGER_ALARM".CLIENT.U1_STA3_COAXIAL.ALARMS.LASER_CALIB_REQUIERED_A;
END_REGION

REGION Network 49: UNIT 01 STATION 3 COAXIAL NEW JET CALIBRATION REQUIERED ALARM
   RUNG wire#powerrail
      { S7_Templates := "SrcType := Int" } EQ_Contact(in1 := "DB16002_U01_STA3_COAXIAL_CLIENT_INTERFACE".U1_STA3_CAM_Read.Variable.Status, in2 := -1)
      Contact( "DB16002_U01_STA3_COAXIAL_CLIENT_INTERFACE".U1_STA3_CAM_Read.Variable.FailedToConnectToCamera )
      wire#w1
      Contact( "DB7254_UNIT_01_STA_3_COAXIAL_ENABLE_DISABLE".ENABLED )
      wire#w2
      Coil( "DB16000_OPC_UA_TRIGGER_ALARM".CLIENT.U1_STA3_COAXIAL.ALARMS.JET_CALIB_REQUIERED_A )
   END_RUNG
   RUNG wire#powerrail
      Contact( "DB16000_OPC_UA_TRIGGER_ALARM".CLIENT.U1_STA3_COAXIAL.ALARMS.JET_CALIB_REQUIERED_A )
      I_Contact( "DB2120_MPP_ITC_IPC".RESET_FAULTS )
   END_RUNG wire#w1
   RUNG wire#w2
      Coil( "DB426_ALARMS_WARNINGS".UNIT_01.STATION_3_COAXIAL."716643" )
   END_RUNG
   // the same network as SCL:
   "DB16000_OPC_UA_TRIGGER_ALARM".CLIENT.U1_STA3_COAXIAL.ALARMS.JET_CALIB_REQUIERED_A := ((("DB16002_U01_STA3_COAXIAL_CLIENT_INTERFACE".U1_STA3_CAM_Read.Variable.Status = (-1)) AND "DB16002_U01_STA3_COAXIAL_CLIENT_INTERFACE".U1_STA3_CAM_Read.Variable.FailedToConnectToCamera) OR ("DB16000_OPC_UA_TRIGGER_ALARM".CLIENT.U1_STA3_COAXIAL.ALARMS.JET_CALIB_REQUIERED_A AND NOT "DB2120_MPP_ITC_IPC".RESET_FAULTS)) AND "DB7254_UNIT_01_STA_3_COAXIAL_ENABLE_DISABLE".ENABLED;
   "DB426_ALARMS_WARNINGS".UNIT_01.STATION_3_COAXIAL."716643" := "DB16000_OPC_UA_TRIGGER_ALARM".CLIENT.U1_STA3_COAXIAL.ALARMS.JET_CALIB_REQUIERED_A;
END_REGION

REGION Network 50: UNIT 01 STATION 3 COAXIAL NEW CLADDING CALIBRBATION REQUIERED ALARM
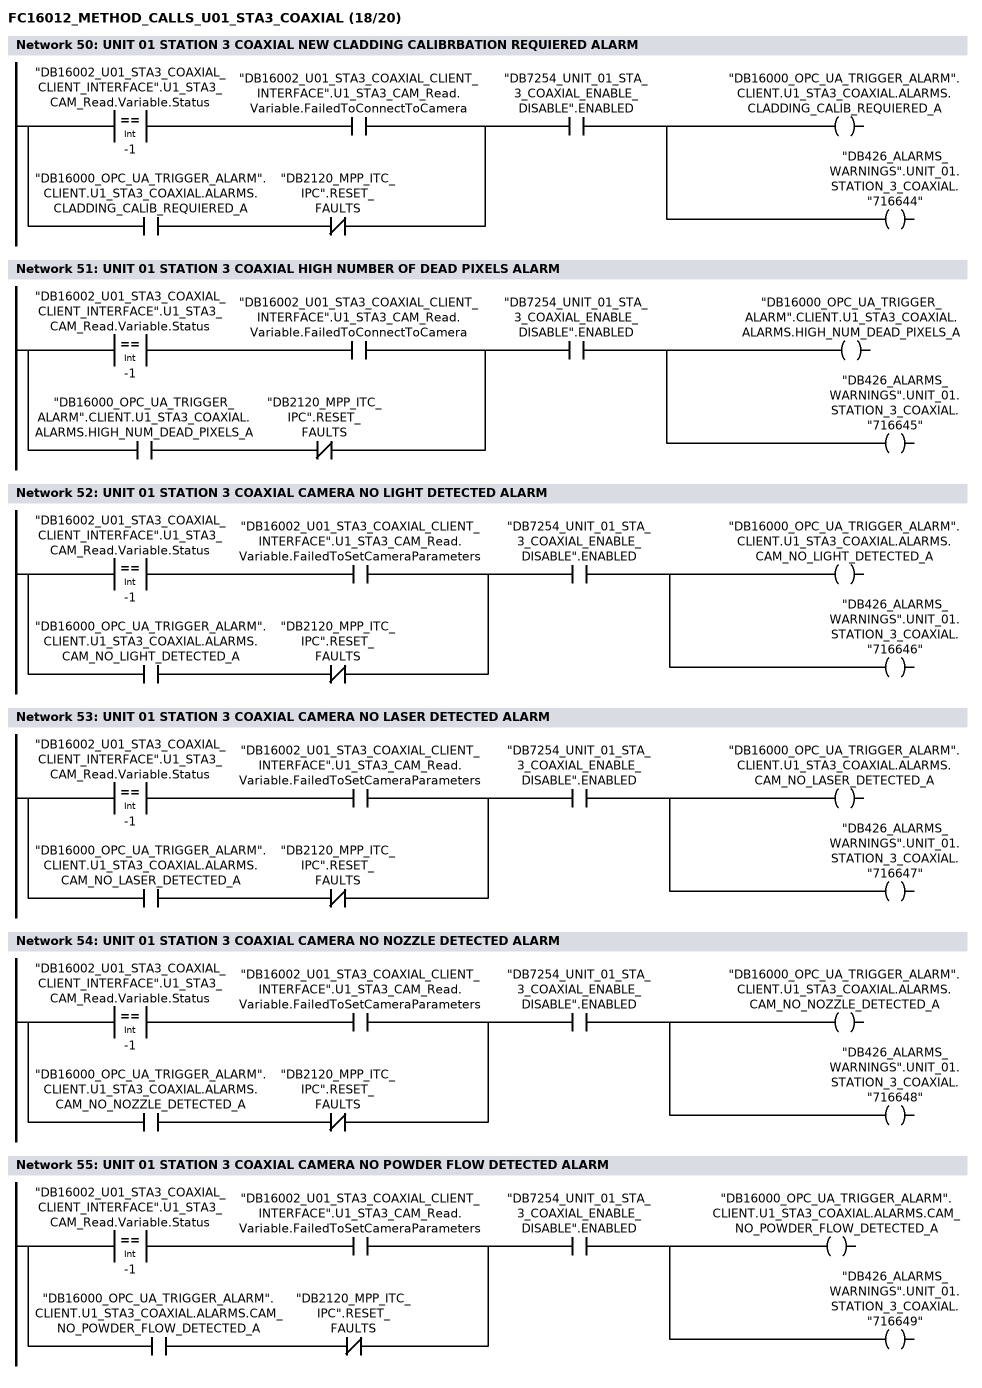
   RUNG wire#powerrail
      { S7_Templates := "SrcType := Int" } EQ_Contact(in1 := "DB16002_U01_STA3_COAXIAL_CLIENT_INTERFACE".U1_STA3_CAM_Read.Variable.Status, in2 := -1)
      Contact( "DB16002_U01_STA3_COAXIAL_CLIENT_INTERFACE".U1_STA3_CAM_Read.Variable.FailedToConnectToCamera )
      wire#w1
      Contact( "DB7254_UNIT_01_STA_3_COAXIAL_ENABLE_DISABLE".ENABLED )
      wire#w2
      Coil( "DB16000_OPC_UA_TRIGGER_ALARM".CLIENT.U1_STA3_COAXIAL.ALARMS.CLADDING_CALIB_REQUIERED_A )
   END_RUNG
   RUNG wire#powerrail
      Contact( "DB16000_OPC_UA_TRIGGER_ALARM".CLIENT.U1_STA3_COAXIAL.ALARMS.CLADDING_CALIB_REQUIERED_A )
      I_Contact( "DB2120_MPP_ITC_IPC".RESET_FAULTS )
   END_RUNG wire#w1
   RUNG wire#w2
      Coil( "DB426_ALARMS_WARNINGS".UNIT_01.STATION_3_COAXIAL."716644" )
   END_RUNG
   // the same network as SCL:
   "DB16000_OPC_UA_TRIGGER_ALARM".CLIENT.U1_STA3_COAXIAL.ALARMS.CLADDING_CALIB_REQUIERED_A := ((("DB16002_U01_STA3_COAXIAL_CLIENT_INTERFACE".U1_STA3_CAM_Read.Variable.Status = (-1)) AND "DB16002_U01_STA3_COAXIAL_CLIENT_INTERFACE".U1_STA3_CAM_Read.Variable.FailedToConnectToCamera) OR ("DB16000_OPC_UA_TRIGGER_ALARM".CLIENT.U1_STA3_COAXIAL.ALARMS.CLADDING_CALIB_REQUIERED_A AND NOT "DB2120_MPP_ITC_IPC".RESET_FAULTS)) AND "DB7254_UNIT_01_STA_3_COAXIAL_ENABLE_DISABLE".ENABLED;
   "DB426_ALARMS_WARNINGS".UNIT_01.STATION_3_COAXIAL."716644" := "DB16000_OPC_UA_TRIGGER_ALARM".CLIENT.U1_STA3_COAXIAL.ALARMS.CLADDING_CALIB_REQUIERED_A;
END_REGION

